LIN {X 0,Y 149.917,Z 380.311,A -85,B 0,C 180,E1 -25491.126,E2 -25491.126} C_VEL
LIN {X 0,Y 151.658,Z 366.446,A -85,B 0,C 180,E1 -25492.001,E2 -25492.001} C_VEL
LIN {X 0,Y 154.477,Z 327.485,A -85,B 0,C 180,E1 -25493.636,E2 -25493.636} C_VEL
LIN {X 0,Y 149.721,Z 315.229,A -85,B 0,C 180,E1 -25495.993,E2 -25495.993} C_VEL
LIN {X 0,Y 144.955,Z 306.325,A -85,B 0,C 180,E1 -25498.361,E2 -25498.361} C_VEL
LIN {X 0,Y 138.94,Z 296.328,A -85,B 0,C 180,E1 -25501.592,E2 -25501.592} C_VEL
LIN {X 0,Y 134.501,Z 289.677,A -85,B 0,C 180,E1 -25504.225,E2 -25504.225} C_VEL
LIN {X 0,Y 131.955,Z 285.984,A -85,B 0,C 180,E1 -25505.867,E2 -25505.867} C_VEL
LIN {X 0,Y 129.466,Z 282.342,A -85,B 0,C 180,E1 -25507.593,E2 -25507.593} C_VEL
LIN {X 0,Y 126.831,Z 279.366,A -85,B 0,C 180,E1 -25509.458,E2 -25509.458} C_VEL
LIN {X 0,Y 125.614,Z 277.233,A -85,B 0,C 180,E1 -25510.449,E2 -25510.449} C_VEL
LIN {X 0,Y 123.042,Z 275.019,A -85,B 0,C 180,E1 -25512.437,E2 -25512.437} C_VEL
LIN {X 0,Y 121.953,Z 272.605,A -85,B 0,C 180,E1 -25513.756,E2 -25513.756} C_VEL
LIN {X 0,Y 121.871,Z 271.831,A -85,B 0,C 180,E1 -25514.986,E2 -25514.986} C_VEL
LIN {X 0,Y 121.84,Z 271.763,A -85,B 0,C 180,E1 -25520.633,E2 -25520.633} C_VEL
LIN {X 0,Y 121.893,Z 271.784,A -85,B 0,C 180,E1 -25524.805,E2 -25524.805} C_VEL
LIN {X 0,Y 121.893,Z 271.751,A -85,B 0,C 180,E1 -25529.871,E2 -25529.871} C_VEL
LIN {X 0,Y 121.974,Z 271.79,A -85,B 0,C 180,E1 -25537.212,E2 -25537.212} C_VEL
LIN {X 0,Y 122.06,Z 271.721,A -85,B 0,C 180,E1 -25543.281,E2 -25543.281} C_VEL
LIN {X 0,Y 122.287,Z 271.749,A -85,B 0,C 180,E1 -25547.702,E2 -25547.702} C_VEL
LIN {X 0,Y 122.391,Z 271.714,A -85,B 0,C 180,E1 -25550.092,E2 -25550.092} C_VEL
LIN {X 0,Y 122.559,Z 271.673,A -85,B 0,C 180,E1 -25556.724,E2 -25556.724} C_VEL
LIN {X 0,Y 123.024,Z 271.658,A -85,B 0,C 180,E1 -25560.011,E2 -25560.011} C_VEL
LIN {X 0,Y 122.411,Z 271.686,A -85,B 0,C 180,E1 -25566.605,E2 -25566.605} C_VEL
LIN {X 0,Y 122.4,Z 271.735,A -85,B 0,C 180,E1 -25569.93,E2 -25569.93} C_VEL
LIN {X 0,Y 122.2,Z 271.727,A -85,B 0,C 180,E1 -25573.311,E2 -25573.311} C_VEL
LIN {X 0,Y 122.035,Z 271.781,A -85,B 0,C 180,E1 -25580.226,E2 -25580.226} C_VEL
LIN {X 0,Y 122.109,Z 271.951,A -85,B 0,C 180,E1 -25582.499,E2 -25582.499} C_VEL
LIN {X 0,Y 122.335,Z 273.222,A -85,B 0,C 180,E1 -25583.623,E2 -25583.623} C_VEL
LIN {X 0,Y 123.788,Z 275.687,A -85,B 0,C 180,E1 -25584.99,E2 -25584.99} C_VEL
LIN {X 0,Y 125.956,Z 277.488,A -85,B 0,C 180,E1 -25586.626,E2 -25586.626} C_VEL
LIN {X 0,Y 127.946,Z 280.764,A -85,B 0,C 180,E1 -25588.186,E2 -25588.186} C_VEL
LIN {X 0,Y 129.741,Z 282.697,A -85,B 0,C 180,E1 -25589.425,E2 -25589.425} C_VEL
LIN {X 0,Y 133.694,Z 288.444,A -85,B 0,C 180,E1 -25592.092,E2 -25592.092} C_VEL
LIN {X 0,Y 138.036,Z 294.974,A -85,B 0,C 180,E1 -25594.722,E2 -25594.722} C_VEL
LIN {X 0,Y 143.351,Z 303.799,A -85,B 0,C 180,E1 -25597.654,E2 -25597.654} C_VEL
LIN {X 0,Y 148.299,Z 314.843,A -85,B 0,C 180,E1 -25600.312,E2 -25600.312} C_VEL
LIN {X 0,Y 153.035,Z 327.628,A -85,B 0,C 180,E1 -25602.751,E2 -25602.751} C_VEL
LIN {X 0,Y 154.24,Z 331.13,A -85,B 0,C 180,E1 -25603.35,E2 -25603.35} C_VEL
LIN {X 0,Y 151.137,Z 374.069,A -85,B 0,C 180,E1 -25605.228,E2 -25605.228} C_VEL
LIN {X 0,Y 149.139,Z 387.318,A -85,B 0,C 180,E1 -25606.198,E2 -25606.198} C_VEL
LIN {X 0,Y 146.572,Z 399.758,A -85,B 0,C 180,E1 -25607.599,E2 -25607.599} C_VEL
LIN {X 0,Y 143.346,Z 411.689,A -85,B 0,C 180,E1 -25609.484,E2 -25609.484} C_VEL
LIN {X 0,Y 139.628,Z 423.169,A -85,B 0,C 180,E1 -25611.93,E2 -25611.93} C_VEL
LIN {X 0,Y 135.702,Z 433.514,A -85,B 0,C 180,E1 -25614.816,E2 -25614.816} C_VEL
LIN {X 0,Y 131.666,Z 443.348,A -85,B 0,C 180,E1 -25618.48,E2 -25618.48} C_VEL
LIN {X 0,Y 128.331,Z 451.168,A -85,B 0,C 180,E1 -25622.255,E2 -25622.255} C_VEL
LIN {X 0,Y 124.933,Z 458.531,A -85,B 0,C 180,E1 -25626.808,E2 -25626.808} C_VEL
LIN {X 0,Y 122.288,Z 464.413,A -85,B 0,C 180,E1 -25631.571,E2 -25631.571} C_VEL
LIN {X 0,Y 120.578,Z 469.032,A -85,B 0,C 180,E1 -25636.515,E2 -25636.515} C_VEL
LIN {X 0,Y 119.827,Z 471.455,A -85,B 0,C 180,E1 -25639.863,E2 -25639.863} C_VEL
LIN {X 0,Y 119.356,Z 473.43,A -85,B 0,C 180,E1 -25643.234,E2 -25643.234} C_VEL
LIN {X 0,Y 119.172,Z 474.984,A -85,B 0,C 180,E1 -25646.616,E2 -25646.616} C_VEL
LIN {X 0,Y 119.252,Z 476.091,A -85,B 0,C 180,E1 -25649.997,E2 -25649.997} C_VEL
LIN {X 0,Y 119.173,Z 476.77,A -85,B 0,C 180,E1 -25653.378,E2 -25653.378} C_VEL
LIN {X 0,Y 119.89,Z 476.987,A -85,B 0,C 180,E1 -25660.126,E2 -25660.126} C_VEL
LIN {X 0,Y 120.731,Z 476.514,A -85,B 0,C 180,E1 -25663.462,E2 -25663.462} C_VEL
LIN {X 0,Y 123.396,Z 474.35,A -85,B 0,C 180,E1 -25669.979,E2 -25669.979} C_VEL
LIN {X 0,Y 126.498,Z 471.676,A -85,B 0,C 180,E1 -25674.622,E2 -25674.622} C_VEL
LIN {X 0,Y 130.853,Z 467.562,A -85,B 0,C 180,E1 -25679.473,E2 -25679.473} C_VEL
LIN {X 0,Y 136.528,Z 461.498,A -85,B 0,C 180,E1 -25684.485,E2 -25684.485} C_VEL
LIN {X 0,Y 141.954,Z 455.109,A -85,B 0,C 180,E1 -25688.23,E2 -25688.23} C_VEL
LIN {X 0,Y 143.742,Z 452.844,A -85,B 0,C 180,E1 -25689.335,E2 -25689.335} C_VEL
LIN {X 0,Y 145.909,Z 449.452,A -85,B 0,C 180,E1 -25691.051,E2 -25691.051} C_VEL
LIN {X 0,Y 148.208,Z 443.627,A -85,B 0,C 180,E1 -25694.05,E2 -25694.05} C_VEL
LIN {X 0,Y 150.646,Z 437.293,A -85,B 0,C 180,E1 -25696.796,E2 -25696.796} C_VEL
LIN {X 0,Y 152.93,Z 433.024,A -85,B 0,C 180,E1 -25698.077,E2 -25698.077} C_VEL
LIN {X 0,Y 158.845,Z 422.424,A -85,B 0,C 180,E1 -25700.238,E2 -25700.238} C_VEL
LIN {X 0,Y 164.023,Z 411.245,A -85,B 0,C 180,E1 -25701.932,E2 -25701.932} C_VEL
LIN {X 0,Y 168.444,Z 399.218,A -85,B 0,C 180,E1 -25703.309,E2 -25703.309} C_VEL
LIN {X 0,Y 171.869,Z 387.049,A -85,B 0,C 180,E1 -25704.268,E2 -25704.268} C_VEL
LIN {X 0,Y 174.526,Z 373.628,A -85,B 0,C 180,E1 -25704.952,E2 -25704.952} C_VEL
LIN {X 0,Y 176.895,Z 350.528,A -85,B 0,C 180,E1 -25705.791,E2 -25705.791} C_VEL
LIN {X 0,Y 174.129,Z 342.792,A -85,B 0,C 180,E1 -25708.604,E2 -25708.604} C_VEL
LIN {X 0,Y 171.468,Z 336.339,A -85,B 0,C 180,E1 -25711.689,E2 -25711.689} C_VEL
LIN {X 0,Y 170.136,Z 333.483,A -85,B 0,C 180,E1 -25713.465,E2 -25713.465} C_VEL
LIN {X 0,Y 168.525,Z 330.627,A -85,B 0,C 180,E1 -25715.864,E2 -25715.864} C_VEL
LIN {X 0,Y 166.557,Z 327.038,A -85,B 0,C 180,E1 -25719.732,E2 -25719.732} C_VEL
LIN {X 0,Y 164.734,Z 324.215,A -85,B 0,C 180,E1 -25727.052,E2 -25727.052} C_VEL
LIN {X 0,Y 164.785,Z 323.798,A -85,B 0,C 180,E1 -25730.169,E2 -25730.169} C_VEL
LIN {X 0,Y 166.586,Z 326.483,A -85,B 0,C 180,E1 -25737.423,E2 -25737.423} C_VEL
LIN {X 0,Y 168.586,Z 330.291,A -85,B 0,C 180,E1 -25741.404,E2 -25741.404} C_VEL
LIN {X 0,Y 170.651,Z 333.974,A -85,B 0,C 180,E1 -25744.408,E2 -25744.408} C_VEL
LIN {X 0,Y 173.991,Z 340.469,A -85,B 0,C 180,E1 -25748.266,E2 -25748.266} C_VEL
LIN {X 0,Y 175.805,Z 344.628,A -85,B 0,C 180,E1 -25750.115,E2 -25750.115} C_VEL
LIN {X 0,Y 177.089,Z 348.243,A -85,B 0,C 180,E1 -25751.363,E2 -25751.363} C_VEL
LIN {X 0,Y 174.518,Z 372.291,A -85,B 0,C 180,E1 -25752.203,E2 -25752.203} C_VEL
LIN {X 0,Y 172.102,Z 384.595,A -85,B 0,C 180,E1 -25752.859,E2 -25752.859} C_VEL
LIN {X 0,Y 168.746,Z 396.829,A -85,B 0,C 180,E1 -25753.859,E2 -25753.859} C_VEL
LIN {X 0,Y 164.693,Z 408.226,A -85,B 0,C 180,E1 -25755.201,E2 -25755.201} C_VEL
LIN {X 0,Y 159.734,Z 419.22,A -85,B 0,C 180,E1 -25756.882,E2 -25756.882} C_VEL
LIN {X 0,Y 154.191,Z 429.462,A -85,B 0,C 180,E1 -25758.962,E2 -25758.962} C_VEL
LIN {X 0,Y 148.873,Z 437.871,A -85,B 0,C 180,E1 -25761.196,E2 -25761.196} C_VEL
LIN {X 0,Y 142.551,Z 446.547,A -85,B 0,C 180,E1 -25764.212,E2 -25764.212} C_VEL
LIN {X 0,Y 136.628,Z 453.681,A -85,B 0,C 180,E1 -25767.565,E2 -25767.565} C_VEL
LIN {X 0,Y 129.941,Z 460.795,A -85,B 0,C 180,E1 -25772.199,E2 -25772.199} C_VEL
LIN {X 0,Y 123.977,Z 466.358,A -85,B 0,C 180,E1 -25777.479,E2 -25777.479} C_VEL
LIN {X 0,Y 119.536,Z 470.003,A -85,B 0,C 180,E1 -25782.704,E2 -25782.704} C_VEL
LIN {X 0,Y 116.059,Z 472.435,A -85,B 0,C 180,E1 -25788.237,E2 -25788.237} C_VEL
LIN {X 0,Y 113.852,Z 473.647,A -85,B 0,C 180,E1 -25793.345,E2 -25793.345} C_VEL
LIN {X 0,Y 112.133,Z 473.944,A -85,B 0,C 180,E1 -25799.911,E2 -25799.911} C_VEL
LIN {X 0,Y 111.656,Z 473.511,A -85,B 0,C 180,E1 -25803.861,E2 -25803.861} C_VEL
LIN {X 0,Y 111.688,Z 471.595,A -85,B 0,C 180,E1 -25810.67,E2 -25810.67} C_VEL
LIN {X 0,Y 112.749,Z 468.214,A -85,B 0,C 180,E1 -25817.402,E2 -25817.402} C_VEL
LIN {X 0,Y 114.461,Z 464.126,A -85,B 0,C 180,E1 -25822.949,E2 -25822.949} C_VEL
LIN {X 0,Y 116.793,Z 458.839,A -85,B 0,C 180,E1 -25828.279,E2 -25828.279} C_VEL
LIN {X 0,Y 120.046,Z 452.098,A -85,B 0,C 180,E1 -25833.359,E2 -25833.359} C_VEL
LIN {X 0,Y 124.034,Z 443.668,A -85,B 0,C 180,E1 -25838.146,E2 -25838.146} C_VEL
LIN {X 0,Y 127.929,Z 435.024,A -85,B 0,C 180,E1 -25841.891,E2 -25841.891} C_VEL
LIN {X 0,Y 131.791,Z 425.809,A -85,B 0,C 180,E1 -25844.967,E2 -25844.967} C_VEL
LIN {X 0,Y 135.727,Z 415.062,A -85,B 0,C 180,E1 -25847.713,E2 -25847.713} C_VEL
LIN {X 0,Y 139.216,Z 403.697,A -85,B 0,C 180,E1 -25849.925,E2 -25849.925} C_VEL
LIN {X 0,Y 142.282,Z 391.091,A -85,B 0,C 180,E1 -25851.746,E2 -25851.746} C_VEL
LIN {X 0,Y 144.771,Z 377.58,A -85,B 0,C 180,E1 -25853.038,E2 -25853.038} C_VEL
LIN {X 0,Y 146.278,Z 364.752,A -85,B 0,C 180,E1 -25853.806,E2 -25853.806} C_VEL
LIN {X 0,Y 148.904,Z 329.221,A -85,B 0,C 180,E1 -25855.326,E2 -25855.326} C_VEL
LIN {X 0,Y 144.595,Z 318.262,A -85,B 0,C 180,E1 -25857.637,E2 -25857.637} C_VEL
LIN {X 0,Y 139.163,Z 308.178,A -85,B 0,C 180,E1 -25860.558,E2 -25860.558} C_VEL
LIN {X 0,Y 133.577,Z 298.915,A -85,B 0,C 180,E1 -25863.891,E2 -25863.891} C_VEL
LIN {X 0,Y 128.421,Z 291.313,A -85,B 0,C 180,E1 -25867.331,E2 -25867.331} C_VEL
LIN {X 0,Y 125.856,Z 287.671,A -85,B 0,C 180,E1 -25869.228,E2 -25869.228} C_VEL
LIN {X 0,Y 123.261,Z 284.164,A -85,B 0,C 180,E1 -25871.279,E2 -25871.279} C_VEL
LIN {X 0,Y 122.402,Z 283.086,A -85,B 0,C 180,E1 -25871.994,E2 -25871.994} C_VEL
LIN {X 0,Y 119.918,Z 280.305,A -85,B 0,C 180,E1 -25874.161,E2 -25874.161} C_VEL
LIN {X 0,Y 118.797,Z 278.232,A -85,B 0,C 180,E1 -25875.317,E2 -25875.317} C_VEL
LIN {X 0,Y 116.391,Z 276.344,A -85,B 0,C 180,E1 -25877.624,E2 -25877.624} C_VEL
LIN {X 0,Y 114.926,Z 273.384,A -85,B 0,C 180,E1 -25879.782,E2 -25879.782} C_VEL
LIN {X 0,Y 114.783,Z 272.721,A -85,B 0,C 180,E1 -25881.144,E2 -25881.144} C_VEL
LIN {X 0,Y 114.795,Z 272.679,A -85,B 0,C 180,E1 -25886.58,E2 -25886.58} C_VEL
LIN {X 0,Y 114.806,Z 272.629,A -85,B 0,C 180,E1 -25890.692,E2 -25890.692} C_VEL
LIN {X 0,Y 114.893,Z 272.673,A -85,B 0,C 180,E1 -25896.576,E2 -25896.576} C_VEL
LIN {X 0,Y 114.963,Z 272.603,A -85,B 0,C 180,E1 -25902.215,E2 -25902.215} C_VEL
LIN {X 0,Y 115.306,Z 272.605,A -85,B 0,C 180,E1 -25909.476,E2 -25909.476} C_VEL
LIN {X 0,Y 115.485,Z 272.55,A -85,B 0,C 180,E1 -25916.523,E2 -25916.523} C_VEL
LIN {X 0,Y 115.976,Z 272.536,A -85,B 0,C 180,E1 -25920.012,E2 -25920.012} C_VEL
LIN {X 0,Y 115.354,Z 272.567,A -85,B 0,C 180,E1 -25927.011,E2 -25927.011} C_VEL
LIN {X 0,Y 115.215,Z 272.604,A -85,B 0,C 180,E1 -25932.572,E2 -25932.572} C_VEL
LIN {X 0,Y 115.072,Z 272.837,A -85,B 0,C 180,E1 -25936.42,E2 -25936.42} C_VEL
LIN {X 0,Y 115.35,Z 274.101,A -85,B 0,C 180,E1 -25937.863,E2 -25937.863} C_VEL
LIN {X 0,Y 116.774,Z 276.567,A -85,B 0,C 180,E1 -25939.571,E2 -25939.571} C_VEL
LIN {X 0,Y 119.245,Z 278.524,A -85,B 0,C 180,E1 -25941.917,E2 -25941.917} C_VEL
LIN {X 0,Y 121.112,Z 281.678,A -85,B 0,C 180,E1 -25943.742,E2 -25943.742} C_VEL
LIN {X 0,Y 123.21,Z 283.867,A -85,B 0,C 180,E1 -25945.482,E2 -25945.482} C_VEL
LIN {X 0,Y 125.712,Z 287.403,A -85,B 0,C 180,E1 -25947.483,E2 -25947.483} C_VEL
LIN {X 0,Y 127.202,Z 289.451,A -85,B 0,C 180,E1 -25948.601,E2 -25948.601} C_VEL
LIN {X 0,Y 130.687,Z 294.469,A -85,B 0,C 180,E1 -25951.05,E2 -25951.05} C_VEL
LIN {X 0,Y 136.464,Z 303.687,A -85,B 0,C 180,E1 -25954.716,E2 -25954.716} C_VEL
LIN {X 0,Y 139.996,Z 310.198,A -85,B 0,C 180,E1 -25956.777,E2 -25956.777} C_VEL
LIN {X 0,Y 145.15,Z 322.701,A -85,B 0,C 180,E1 -25959.72,E2 -25959.72} C_VEL
LIN {X 0,Y 148.753,Z 333.117,A -85,B 0,C 180,E1 -25961.715,E2 -25961.715} C_VEL
LIN {X 0,Y 145.583,Z 374.151,A -85,B 0,C 180,E1 -25963.534,E2 -25963.534} C_VEL
LIN {X 0,Y 143.513,Z 387.259,A -85,B 0,C 180,E1 -25964.506,E2 -25964.506} C_VEL
LIN {X 0,Y 140.849,Z 399.691,A -85,B 0,C 180,E1 -25965.934,E2 -25965.934} C_VEL
LIN {X 0,Y 137.486,Z 411.614,A -85,B 0,C 180,E1 -25967.859,E2 -25967.859} C_VEL
LIN {X 0,Y 133.601,Z 423.09,A -85,B 0,C 180,E1 -25970.367,E2 -25970.367} C_VEL
LIN {X 0,Y 129.491,Z 433.431,A -85,B 0,C 180,E1 -25973.341,E2 -25973.341} C_VEL
LIN {X 0,Y 125.432,Z 442.85,A -85,B 0,C 180,E1 -25976.955,E2 -25976.955} C_VEL
LIN {X 0,Y 122.059,Z 450.396,A -85,B 0,C 180,E1 -25980.695,E2 -25980.695} C_VEL
LIN {X 0,Y 118.421,Z 457.879,A -85,B 0,C 180,E1 -25985.451,E2 -25985.451} C_VEL
LIN {X 0,Y 115.537,Z 463.867,A -85,B 0,C 180,E1 -25990.451,E2 -25990.451} C_VEL
LIN {X 0,Y 113.667,Z 468.589,A -85,B 0,C 180,E1 -25995.678,E2 -25995.678} C_VEL
LIN {X 0,Y 112.514,Z 472.165,A -85,B 0,C 180,E1 -26001.013,E2 -26001.013} C_VEL
LIN {X 0,Y 112.08,Z 474.707,A -85,B 0,C 180,E1 -26006.402,E2 -26006.402} C_VEL
LIN {X 0,Y 112.156,Z 475.888,A -85,B 0,C 180,E1 -26009.997,E2 -26009.997} C_VEL
LIN {X 0,Y 112.081,Z 476.612,A -85,B 0,C 180,E1 -26013.592,E2 -26013.592} C_VEL
LIN {X 0,Y 112.902,Z 476.907,A -85,B 0,C 180,E1 -26020.76,E2 -26020.76} C_VEL
LIN {X 0,Y 113.812,Z 476.49,A -85,B 0,C 180,E1 -26024.297,E2 -26024.297} C_VEL
LIN {X 0,Y 115.101,Z 475.666,A -85,B 0,C 180,E1 -26027.773,E2 -26027.773} C_VEL
LIN {X 0,Y 116.721,Z 474.438,A -85,B 0,C 180,E1 -26031.175,E2 -26031.175} C_VEL
LIN {X 0,Y 121.378,Z 470.796,A -85,B 0,C 180,E1 -26037.591,E2 -26037.591} C_VEL
LIN {X 0,Y 125.754,Z 466.888,A -85,B 0,C 180,E1 -26042.064,E2 -26042.064} C_VEL
LIN {X 0,Y 130.741,Z 461.895,A -85,B 0,C 180,E1 -26046.246,E2 -26046.246} C_VEL
LIN {X 0,Y 136.461,Z 455.652,A -85,B 0,C 180,E1 -26050.07,E2 -26050.07} C_VEL
LIN {X 0,Y 142.8,Z 447.875,A -85,B 0,C 180,E1 -26053.549,E2 -26053.549} C_VEL
LIN {X 0,Y 149.607,Z 438.265,A -85,B 0,C 180,E1 -26056.726,E2 -26056.726} C_VEL
LIN {X 0,Y 152.93,Z 433.024,A -85,B 0,C 180,E1 -26058.077,E2 -26058.077} C_VEL
LIN {X 0,Y 155.209,Z 428.626,A -85,B 0,C 180,E1 -26059.282,E2 -26059.282} C_VEL
LIN {X 0,Y 157.669,Z 421.297,A -85,B 0,C 180,E1 -26061.563,E2 -26061.563} C_VEL
LIN {X 0,Y 159.898,Z 413.531,A -85,B 0,C 180,E1 -26063.626,E2 -26063.626} C_VEL
LIN {X 0,Y 161.717,Z 408.455,A -85,B 0,C 180,E1 -26064.475,E2 -26064.475} C_VEL
LIN {X 0,Y 166.123,Z 396.063,A -85,B 0,C 180,E1 -26065.754,E2 -26065.754} C_VEL
LIN {X 0,Y 169.642,Z 383.168,A -85,B 0,C 180,E1 -26066.625,E2 -26066.625} C_VEL
LIN {X 0,Y 171.89,Z 370.23,A -85,B 0,C 180,E1 -26067.222,E2 -26067.222} C_VEL
LIN {X 0,Y 173.598,Z 353.693,A -85,B 0,C 180,E1 -26067.801,E2 -26067.801} C_VEL
LIN {X 0,Y 171.078,Z 346.284,A -85,B 0,C 180,E1 -26070.757,E2 -26070.757} C_VEL
LIN {X 0,Y 168.825,Z 340.5,A -85,B 0,C 180,E1 -26073.847,E2 -26073.847} C_VEL
LIN {X 0,Y 166.972,Z 337.147,A -85,B 0,C 180,E1 -26076.764,E2 -26076.764} C_VEL
LIN {X 0,Y 165.208,Z 333.639,A -85,B 0,C 180,E1 -26080.684,E2 -26080.684} C_VEL
LIN {X 0,Y 163.761,Z 331.034,A -85,B 0,C 180,E1 -26087.988,E2 -26087.988} C_VEL
LIN {X 0,Y 163.867,Z 331.008,A -85,B 0,C 180,E1 -26090.536,E2 -26090.536} C_VEL
LIN {X 0,Y 165.36,Z 333.254,A -85,B 0,C 180,E1 -26096.778,E2 -26096.778} C_VEL
LIN {X 0,Y 167.707,Z 337.979,A -85,B 0,C 180,E1 -26101.628,E2 -26101.628} C_VEL
LIN {X 0,Y 169.661,Z 341.982,A -85,B 0,C 180,E1 -26104.537,E2 -26104.537} C_VEL
LIN {X 0,Y 172.173,Z 347.158,A -85,B 0,C 180,E1 -26107.552,E2 -26107.552} C_VEL
LIN {X 0,Y 173.612,Z 350.795,A -85,B 0,C 180,E1 -26109.135,E2 -26109.135} C_VEL
LIN {X 0,Y 173.827,Z 351.507,A -85,B 0,C 180,E1 -26109.379,E2 -26109.379} C_VEL
LIN {X 0,Y 171.331,Z 373.134,A -85,B 0,C 180,E1 -26110.122,E2 -26110.122} C_VEL
LIN {X 0,Y 168.814,Z 385.293,A -85,B 0,C 180,E1 -26110.767,E2 -26110.767} C_VEL
LIN {X 0,Y 165.125,Z 397.939,A -85,B 0,C 180,E1 -26111.798,E2 -26111.798} C_VEL
LIN {X 0,Y 160.24,Z 410.64,A -85,B 0,C 180,E1 -26113.311,E2 -26113.311} C_VEL
LIN {X 0,Y 154.705,Z 422.04,A -85,B 0,C 180,E1 -26115.137,E2 -26115.137} C_VEL
LIN {X 0,Y 148.822,Z 431.947,A -85,B 0,C 180,E1 -26117.249,E2 -26117.249} C_VEL
LIN {X 0,Y 142.118,Z 441.572,A -85,B 0,C 180,E1 -26120.026,E2 -26120.026} C_VEL
LIN {X 0,Y 135.661,Z 449.573,A -85,B 0,C 180,E1 -26123.148,E2 -26123.148} C_VEL
LIN {X 0,Y 129.633,Z 456.128,A -85,B 0,C 180,E1 -26126.598,E2 -26126.598} C_VEL
LIN {X 0,Y 123.154,Z 462.318,A -85,B 0,C 180,E1 -26131.135,E2 -26131.135} C_VEL
LIN {X 0,Y 117.771,Z 466.853,A -85,B 0,C 180,E1 -26135.857,E2 -26135.857} C_VEL
LIN {X 0,Y 112.809,Z 470.549,A -85,B 0,C 180,E1 -26141.622,E2 -26141.622} C_VEL
LIN {X 0,Y 110.245,Z 472.203,A -85,B 0,C 180,E1 -26145.478,E2 -26145.478} C_VEL
LIN {X 0,Y 107.155,Z 473.743,A -85,B 0,C 180,E1 -26151.887,E2 -26151.887} C_VEL
LIN {X 0,Y 105.413,Z 474.1,A -85,B 0,C 180,E1 -26157.771,E2 -26157.771} C_VEL
LIN {X 0,Y 104.727,Z 473.762,A -85,B 0,C 180,E1 -26161.985,E2 -26161.985} C_VEL
LIN {X 0,Y 104.415,Z 472.99,A -85,B 0,C 180,E1 -26166.185,E2 -26166.185} C_VEL
LIN {X 0,Y 104.572,Z 471.717,A -85,B 0,C 180,E1 -26170.368,E2 -26170.368} C_VEL
LIN {X 0,Y 105.399,Z 468.945,A -85,B 0,C 180,E1 -26176.507,E2 -26176.507} C_VEL
LIN {X 0,Y 107.079,Z 465.06,A -85,B 0,C 180,E1 -26182.46,E2 -26182.46} C_VEL
LIN {X 0,Y 109.414,Z 459.992,A -85,B 0,C 180,E1 -26188.163,E2 -26188.163} C_VEL
LIN {X 0,Y 112.68,Z 453.558,A -85,B 0,C 180,E1 -26193.579,E2 -26193.579} C_VEL
LIN {X 0,Y 116.748,Z 445.487,A -85,B 0,C 180,E1 -26198.658,E2 -26198.658} C_VEL
LIN {X 0,Y 120.75,Z 437.176,A -85,B 0,C 180,E1 -26202.61,E2 -26202.61} C_VEL
LIN {X 0,Y 125.314,Z 426.978,A -85,B 0,C 180,E1 -26206.288,E2 -26206.288} C_VEL
LIN {X 0,Y 129.266,Z 416.931,A -85,B 0,C 180,E1 -26209.042,E2 -26209.042} C_VEL
LIN {X 0,Y 132.911,Z 405.988,A -85,B 0,C 180,E1 -26211.32,E2 -26211.32} C_VEL
LIN {X 0,Y 136.328,Z 392.896,A -85,B 0,C 180,E1 -26213.35,E2 -26213.35} C_VEL
LIN {X 0,Y 138.914,Z 380.37,A -85,B 0,C 180,E1 -26214.66,E2 -26214.66} C_VEL
LIN {X 0,Y 140.641,Z 367.677,A -85,B 0,C 180,E1 -26215.508,E2 -26215.508} C_VEL
LIN {X 0,Y 143.513,Z 331.247,A -85,B 0,C 180,E1 -26217.109,E2 -26217.109} C_VEL
LIN {X 0,Y 139.947,Z 322.152,A -85,B 0,C 180,E1 -26219.157,E2 -26219.157} C_VEL
LIN {X 0,Y 134.956,Z 312.647,A -85,B 0,C 180,E1 -26222.07,E2 -26222.07} C_VEL
LIN {X 0,Y 129.746,Z 303.794,A -85,B 0,C 180,E1 -26225.431,E2 -26225.431} C_VEL
LIN {X 0,Y 125.285,Z 296.99,A -85,B 0,C 180,E1 -26228.634,E2 -26228.634} C_VEL
LIN {X 0,Y 122.561,Z 293.159,A -85,B 0,C 180,E1 -26230.785,E2 -26230.785} C_VEL
LIN {X 0,Y 119.742,Z 289.21,A -85,B 0,C 180,E1 -26233.239,E2 -26233.239} C_VEL
LIN {X 0,Y 117.208,Z 286.087,A -85,B 0,C 180,E1 -26235.636,E2 -26235.636} C_VEL
LIN {X 0,Y 116.356,Z 284.597,A -85,B 0,C 180,E1 -26236.561,E2 -26236.561} C_VEL
LIN {X 0,Y 113.858,Z 282.238,A -85,B 0,C 180,E1 -26239.18,E2 -26239.18} C_VEL
LIN {X 0,Y 112.264,Z 279.369,A -85,B 0,C 180,E1 -26241.26,E2 -26241.26} C_VEL
LIN {X 0,Y 109.315,Z 277.263,A -85,B 0,C 180,E1 -26245.196,E2 -26245.196} C_VEL
LIN {X 0,Y 107.91,Z 274.351,A -85,B 0,C 180,E1 -26248.162,E2 -26248.162} C_VEL
LIN {X 0,Y 107.764,Z 273.577,A -85,B 0,C 180,E1 -26250.733,E2 -26250.733} C_VEL
LIN {X 0,Y 107.861,Z 273.548,A -85,B 0,C 180,E1 -26257.001,E2 -26257.001} C_VEL
LIN {X 0,Y 107.858,Z 273.491,A -85,B 0,C 180,E1 -26261,E2 -26261} C_VEL
LIN {X 0,Y 108.224,Z 273.498,A -85,B 0,C 180,E1 -26268.779,E2 -26268.779} C_VEL
LIN {X 0,Y 108.287,Z 273.437,A -85,B 0,C 180,E1 -26272.555,E2 -26272.555} C_VEL
LIN {X 0,Y 108.902,Z 273.416,A -85,B 0,C 180,E1 -26280.013,E2 -26280.013} C_VEL
LIN {X 0,Y 108.293,Z 273.656,A -85,B 0,C 180,E1 -26287.939,E2 -26287.939} C_VEL
LIN {X 0,Y 108.611,Z 274.943,A -85,B 0,C 180,E1 -26290.145,E2 -26290.145} C_VEL
LIN {X 0,Y 110.026,Z 277.458,A -85,B 0,C 180,E1 -26292.608,E2 -26292.608} C_VEL
LIN {X 0,Y 112.693,Z 279.681,A -85,B 0,C 180,E1 -26296.078,E2 -26296.078} C_VEL
LIN {X 0,Y 114.499,Z 282.825,A -85,B 0,C 180,E1 -26298.347,E2 -26298.347} C_VEL
LIN {X 0,Y 116.809,Z 284.994,A -85,B 0,C 180,E1 -26300.712,E2 -26300.712} C_VEL
LIN {X 0,Y 119.069,Z 288.379,A -85,B 0,C 180,E1 -26302.976,E2 -26302.976} C_VEL
LIN {X 0,Y 120.476,Z 289.98,A -85,B 0,C 180,E1 -26304.227,E2 -26304.227} C_VEL
LIN {X 0,Y 124.461,Z 295.65,A -85,B 0,C 180,E1 -26307.542,E2 -26307.542} C_VEL
LIN {X 0,Y 128.367,Z 301.526,A -85,B 0,C 180,E1 -26310.437,E2 -26310.437} C_VEL
LIN {X 0,Y 134.288,Z 311.608,A -85,B 0,C 180,E1 -26314.361,E2 -26314.361} C_VEL
LIN {X 0,Y 138.192,Z 320.508,A -85,B 0,C 180,E1 -26316.82,E2 -26316.82} C_VEL
LIN {X 0,Y 142.503,Z 332.46,A -85,B 0,C 180,E1 -26319.429,E2 -26319.429} C_VEL
LIN {X 0,Y 143.327,Z 334.933,A -85,B 0,C 180,E1 -26319.918,E2 -26319.918} C_VEL
LIN {X 0,Y 140.209,Z 373.782,A -85,B 0,C 180,E1 -26321.673,E2 -26321.673} C_VEL
LIN {X 0,Y 138.023,Z 387.2,A -85,B 0,C 180,E1 -26322.678,E2 -26322.678} C_VEL
LIN {X 0,Y 135.254,Z 399.624,A -85,B 0,C 180,E1 -26324.131,E2 -26324.131} C_VEL
LIN {X 0,Y 131.733,Z 411.534,A -85,B 0,C 180,E1 -26326.085,E2 -26326.085} C_VEL
LIN {X 0,Y 127.682,Z 423.01,A -85,B 0,C 180,E1 -26328.658,E2 -26328.658} C_VEL
LIN {X 0,Y 123.379,Z 433.349,A -85,B 0,C 180,E1 -26331.719,E2 -26331.719} C_VEL
LIN {X 0,Y 118.769,Z 443.47,A -85,B 0,C 180,E1 -26335.794,E2 -26335.794} C_VEL
LIN {X 0,Y 114.45,Z 452.358,A -85,B 0,C 180,E1 -26340.574,E2 -26340.574} C_VEL
LIN {X 0,Y 110.854,Z 459.428,A -85,B 0,C 180,E1 -26345.661,E2 -26345.661} C_VEL
LIN {X 0,Y 108.031,Z 465.061,A -85,B 0,C 180,E1 -26351.015,E2 -26351.015} C_VEL
LIN {X 0,Y 106.277,Z 469.482,A -85,B 0,C 180,E1 -26356.614,E2 -26356.614} C_VEL
LIN {X 0,Y 105.255,Z 472.793,A -85,B 0,C 180,E1 -26362.323,E2 -26362.323} C_VEL
LIN {X 0,Y 104.985,Z 474.427,A -85,B 0,C 180,E1 -26366.158,E2 -26366.158} C_VEL
LIN {X 0,Y 105.055,Z 475.655,A -85,B 0,C 180,E1 -26369.997,E2 -26369.997} C_VEL
LIN {X 0,Y 104.986,Z 476.452,A -85,B 0,C 180,E1 -26373.835,E2 -26373.835} C_VEL
LIN {X 0,Y 105.915,Z 476.829,A -85,B 0,C 180,E1 -26381.479,E2 -26381.479} C_VEL
LIN {X 0,Y 108.334,Z 475.706,A -85,B 0,C 180,E1 -26388.924,E2 -26388.924} C_VEL
LIN {X 0,Y 110.107,Z 474.534,A -85,B 0,C 180,E1 -26392.515,E2 -26392.515} C_VEL
LIN {X 0,Y 115.138,Z 470.981,A -85,B 0,C 180,E1 -26399.226,E2 -26399.226} C_VEL
LIN {X 0,Y 119.781,Z 467.17,A -85,B 0,C 180,E1 -26403.872,E2 -26403.872} C_VEL
LIN {X 0,Y 125.091,Z 462.291,A -85,B 0,C 180,E1 -26408.167,E2 -26408.167} C_VEL
LIN {X 0,Y 131.132,Z 456.187,A -85,B 0,C 180,E1 -26412.058,E2 -26412.058} C_VEL
LIN {X 0,Y 137.784,Z 448.626,A -85,B 0,C 180,E1 -26415.566,E2 -26415.566} C_VEL
LIN {X 0,Y 144.87,Z 439.188,A -85,B 0,C 180,E1 -26418.755,E2 -26418.755} C_VEL
LIN {X 0,Y 151.249,Z 429.466,A -85,B 0,C 180,E1 -26421.102,E2 -26421.102} C_VEL
LIN {X 0,Y 157.127,Z 418.663,A -85,B 0,C 180,E1 -26423.08,E2 -26423.08} C_VEL
LIN {X 0,Y 161.717,Z 408.455,A -85,B 0,C 180,E1 -26424.475,E2 -26424.475} C_VEL
LIN {X 0,Y 163.43,Z 403.268,A -85,B 0,C 180,E1 -26425.266,E2 -26425.266} C_VEL
LIN {X 0,Y 165.088,Z 394.763,A -85,B 0,C 180,E1 -26426.96,E2 -26426.96} C_VEL
LIN {X 0,Y 166.36,Z 386.008,A -85,B 0,C 180,E1 -26428.476,E2 -26428.476} C_VEL
LIN {X 0,Y 167.38,Z 380.412,A -85,B 0,C 180,E1 -26428.985,E2 -26428.985} C_VEL
LIN {X 0,Y 169.547,Z 366.781,A -85,B 0,C 180,E1 -26429.555,E2 -26429.555} C_VEL
LIN {X 0,Y 170.546,Z 357.001,A -85,B 0,C 180,E1 -26429.892,E2 -26429.892} C_VEL
LIN {X 0,Y 168.536,Z 350.777,A -85,B 0,C 180,E1 -26432.604,E2 -26432.604} C_VEL
LIN {X 0,Y 166.955,Z 346.463,A -85,B 0,C 180,E1 -26435.097,E2 -26435.097} C_VEL
LIN {X 0,Y 165.551,Z 343.752,A -85,B 0,C 180,E1 -26437.53,E2 -26437.53} C_VEL
LIN {X 0,Y 164.009,Z 340.434,A -85,B 0,C 180,E1 -26441.341,E2 -26441.341} C_VEL
LIN {X 0,Y 162.822,Z 337.948,A -85,B 0,C 180,E1 -26448.753,E2 -26448.753} C_VEL
LIN {X 0,Y 162.918,Z 338.115,A -85,B 0,C 180,E1 -26450.48,E2 -26450.48} C_VEL
LIN {X 0,Y 164.244,Z 340.322,A -85,B 0,C 180,E1 -26456.414,E2 -26456.414} C_VEL
LIN {X 0,Y 166.289,Z 344.697,A -85,B 0,C 180,E1 -26460.967,E2 -26460.967} C_VEL
LIN {X 0,Y 167.935,Z 348.304,A -85,B 0,C 180,E1 -26463.611,E2 -26463.611} C_VEL
LIN {X 0,Y 170.15,Z 353.271,A -85,B 0,C 180,E1 -26466.543,E2 -26466.543} C_VEL
LIN {X 0,Y 170.77,Z 354.801,A -85,B 0,C 180,E1 -26467.281,E2 -26467.281} C_VEL
LIN {X 0,Y 168.473,Z 373.679,A -85,B 0,C 180,E1 -26467.938,E2 -26467.938} C_VEL
LIN {X 0,Y 165.927,Z 385.466,A -85,B 0,C 180,E1 -26468.535,E2 -26468.535} C_VEL
LIN {X 0,Y 162.607,Z 396.684,A -85,B 0,C 180,E1 -26469.403,E2 -26469.403} C_VEL
LIN {X 0,Y 158.278,Z 408.082,A -85,B 0,C 180,E1 -26470.661,E2 -26470.661} C_VEL
LIN {X 0,Y 152.842,Z 419.313,A -85,B 0,C 180,E1 -26472.293,E2 -26472.293} C_VEL
LIN {X 0,Y 146.346,Z 430.308,A -85,B 0,C 180,E1 -26474.439,E2 -26474.439} C_VEL
LIN {X 0,Y 139.623,Z 439.826,A -85,B 0,C 180,E1 -26476.996,E2 -26476.996} C_VEL
LIN {X 0,Y 132.749,Z 448.122,A -85,B 0,C 180,E1 -26480.003,E2 -26480.003} C_VEL
LIN {X 0,Y 125.666,Z 455.547,A -85,B 0,C 180,E1 -26483.713,E2 -26483.713} C_VEL
LIN {X 0,Y 118.602,Z 461.98,A -85,B 0,C 180,E1 -26488.284,E2 -26488.284} C_VEL
LIN {X 0,Y 112.947,Z 466.461,A -85,B 0,C 180,E1 -26492.864,E2 -26492.864} C_VEL
LIN {X 0,Y 107.657,Z 470.126,A -85,B 0,C 180,E1 -26498.435,E2 -26498.435} C_VEL
LIN {X 0,Y 104.707,Z 471.896,A -85,B 0,C 180,E1 -26502.416,E2 -26502.416} C_VEL
LIN {X 0,Y 102.221,Z 473.171,A -85,B 0,C 180,E1 -26506.57,E2 -26506.57} C_VEL
LIN {X 0,Y 100.291,Z 473.915,A -85,B 0,C 180,E1 -26510.904,E2 -26510.904} C_VEL
LIN {X 0,Y 98.843,Z 474.208,A -85,B 0,C 180,E1 -26515.336,E2 -26515.336} C_VEL
LIN {X 0,Y 97.913,Z 474.011,A -85,B 0,C 180,E1 -26519.842,E2 -26519.842} C_VEL
LIN {X 0,Y 97.379,Z 473.332,A -85,B 0,C 180,E1 -26524.344,E2 -26524.344} C_VEL
LIN {X 0,Y 97.402,Z 471.953,A -85,B 0,C 180,E1 -26529.673,E2 -26529.673} C_VEL
LIN {X 0,Y 98.068,Z 469.638,A -85,B 0,C 180,E1 -26535.477,E2 -26535.477} C_VEL
LIN {X 0,Y 99.662,Z 465.963,A -85,B 0,C 180,E1 -26541.896,E2 -26541.896} C_VEL
LIN {X 0,Y 102.025,Z 461.105,A -85,B 0,C 180,E1 -26548.029,E2 -26548.029} C_VEL
LIN {X 0,Y 105.703,Z 454.2,A -85,B 0,C 180,E1 -26554.391,E2 -26554.391} C_VEL
LIN {X 0,Y 109.501,Z 447.149,A -85,B 0,C 180,E1 -26559.236,E2 -26559.236} C_VEL
LIN {X 0,Y 113.589,Z 439.211,A -85,B 0,C 180,E1 -26563.419,E2 -26563.419} C_VEL
LIN {X 0,Y 118.28,Z 429.452,A -85,B 0,C 180,E1 -26567.286,E2 -26567.286} C_VEL
LIN {X 0,Y 122.861,Z 418.568,A -85,B 0,C 180,E1 -26570.513,E2 -26570.513} C_VEL
LIN {X 0,Y 126.654,Z 408.057,A -85,B 0,C 180,E1 -26572.859,E2 -26572.859} C_VEL
LIN {X 0,Y 130.245,Z 395.609,A -85,B 0,C 180,E1 -26574.936,E2 -26574.936} C_VEL
LIN {X 0,Y 133.235,Z 382.25,A -85,B 0,C 180,E1 -26576.454,E2 -26576.454} C_VEL
LIN {X 0,Y 135.1,Z 369.805,A -85,B 0,C 180,E1 -26577.395,E2 -26577.395} C_VEL
LIN {X 0,Y 138.27,Z 333.542,A -85,B 0,C 180,E1 -26578.969,E2 -26578.969} C_VEL
LIN {X 0,Y 135.474,Z 326.163,A -85,B 0,C 180,E1 -26580.731,E2 -26580.731} C_VEL
LIN {X 0,Y 129.962,Z 315.474,A -85,B 0,C 180,E1 -26584.266,E2 -26584.266} C_VEL
LIN {X 0,Y 124.778,Z 306.612,A -85,B 0,C 180,E1 -26587.972,E2 -26587.972} C_VEL
LIN {X 0,Y 120.044,Z 299.407,A -85,B 0,C 180,E1 -26591.845,E2 -26591.845} C_VEL
LIN {X 0,Y 116.952,Z 295.13,A -85,B 0,C 180,E1 -26594.699,E2 -26594.699} C_VEL
LIN {X 0,Y 114.24,Z 291.332,A -85,B 0,C 180,E1 -26597.542,E2 -26597.542} C_VEL
LIN {X 0,Y 111.141,Z 287.648,A -85,B 0,C 180,E1 -26601.177,E2 -26601.177} C_VEL
LIN {X 0,Y 110.283,Z 285.967,A -85,B 0,C 180,E1 -26602.424,E2 -26602.424} C_VEL
LIN {X 0,Y 107.59,Z 283.83,A -85,B 0,C 180,E1 -26606.29,E2 -26606.29} C_VEL
LIN {X 0,Y 105.837,Z 280.608,A -85,B 0,C 180,E1 -26609.689,E2 -26609.689} C_VEL
LIN {X 0,Y 101.383,Z 275.635,A -85,B 0,C 180,E1 -26627.486,E2 -26627.486} C_VEL
LIN {X 0,Y 101.665,Z 275.97,A -85,B 0,C 180,E1 -26633.564,E2 -26633.564} C_VEL
LIN {X 0,Y 103.169,Z 277.726,A -85,B 0,C 180,E1 -26640.501,E2 -26640.501} C_VEL
LIN {X 0,Y 105.175,Z 279.877,A -85,B 0,C 180,E1 -26645.765,E2 -26645.765} C_VEL
LIN {X 0,Y 106.478,Z 280.805,A -85,B 0,C 180,E1 -26648.243,E2 -26648.243} C_VEL
LIN {X 0,Y 108.232,Z 283.969,A -85,B 0,C 180,E1 -26651.46,E2 -26651.46} C_VEL
LIN {X 0,Y 110.622,Z 286.247,A -85,B 0,C 180,E1 -26654.844,E2 -26654.844} C_VEL
LIN {X 0,Y 112.595,Z 289.454,A -85,B 0,C 180,E1 -26657.449,E2 -26657.449} C_VEL
LIN {X 0,Y 114.391,Z 291.262,A -85,B 0,C 180,E1 -26659.411,E2 -26659.411} C_VEL
LIN {X 0,Y 116.892,Z 294.871,A -85,B 0,C 180,E1 -26662.047,E2 -26662.047} C_VEL
LIN {X 0,Y 118.727,Z 297.497,A -85,B 0,C 180,E1 -26663.797,E2 -26663.797} C_VEL
LIN {X 0,Y 121.677,Z 301.757,A -85,B 0,C 180,E1 -26666.373,E2 -26666.373} C_VEL
LIN {X 0,Y 125.548,Z 307.938,A -85,B 0,C 180,E1 -26669.447,E2 -26669.447} C_VEL
LIN {X 0,Y 130.814,Z 317.287,A -85,B 0,C 180,E1 -26673.152,E2 -26673.152} C_VEL
LIN {X 0,Y 135.089,Z 328.041,A -85,B 0,C 180,E1 -26676.078,E2 -26676.078} C_VEL
LIN {X 0,Y 138.05,Z 336.95,A -85,B 0,C 180,E1 -26678.028,E2 -26678.028} C_VEL
LIN {X 0,Y 134.945,Z 373.646,A -85,B 0,C 180,E1 -26679.703,E2 -26679.703} C_VEL
LIN {X 0,Y 132.598,Z 387.411,A -85,B 0,C 180,E1 -26680.744,E2 -26680.744} C_VEL
LIN {X 0,Y 129.805,Z 399.422,A -85,B 0,C 180,E1 -26682.174,E2 -26682.174} C_VEL
LIN {X 0,Y 126.121,Z 411.354,A -85,B 0,C 180,E1 -26684.152,E2 -26684.152} C_VEL
LIN {X 0,Y 121.888,Z 422.846,A -85,B 0,C 180,E1 -26686.784,E2 -26686.784} C_VEL
LIN {X 0,Y 117.83,Z 432.119,A -85,B 0,C 180,E1 -26689.557,E2 -26689.557} C_VEL
LIN {X 0,Y 113.703,Z 440.973,A -85,B 0,C 180,E1 -26693.048,E2 -26693.048} C_VEL
LIN {X 0,Y 109.731,Z 448.831,A -85,B 0,C 180,E1 -26697.056,E2 -26697.056} C_VEL
LIN {X 0,Y 105.587,Z 456.531,A -85,B 0,C 180,E1 -26702.226,E2 -26702.226} C_VEL
LIN {X 0,Y 102.222,Z 462.738,A -85,B 0,C 180,E1 -26707.778,E2 -26707.778} C_VEL
LIN {X 0,Y 99.898,Z 467.656,A -85,B 0,C 180,E1 -26713.652,E2 -26713.652} C_VEL
LIN {X 0,Y 98.501,Z 471.419,A -85,B 0,C 180,E1 -26719.722,E2 -26719.722} C_VEL
LIN {X 0,Y 97.913,Z 474.134,A -85,B 0,C 180,E1 -26725.881,E2 -26725.881} C_VEL
LIN {X 0,Y 97.962,Z 475.405,A -85,B 0,C 180,E1 -26729.997,E2 -26729.997} C_VEL
LIN {X 0,Y 97.914,Z 476.266,A -85,B 0,C 180,E1 -26734.113,E2 -26734.113} C_VEL
LIN {X 0,Y 98.227,Z 476.708,A -85,B 0,C 180,E1 -26738.224,E2 -26738.224} C_VEL
LIN {X 0,Y 100.088,Z 476.421,A -85,B 0,C 180,E1 -26746.309,E2 -26746.309} C_VEL
LIN {X 0,Y 103.563,Z 474.627,A -85,B 0,C 180,E1 -26754.024,E2 -26754.024} C_VEL
LIN {X 0,Y 109.006,Z 471.18,A -85,B 0,C 180,E1 -26761.046,E2 -26761.046} C_VEL
LIN {X 0,Y 113.948,Z 467.483,A -85,B 0,C 180,E1 -26765.865,E2 -26765.865} C_VEL
LIN {X 0,Y 119.597,Z 462.717,A -85,B 0,C 180,E1 -26770.267,E2 -26770.267} C_VEL
LIN {X 0,Y 127.087,Z 455.63,A -85,B 0,C 180,E1 -26774.832,E2 -26774.832} C_VEL
LIN {X 0,Y 134.162,Z 447.919,A -85,B 0,C 180,E1 -26778.282,E2 -26778.282} C_VEL
LIN {X 0,Y 140.328,Z 440.113,A -85,B 0,C 180,E1 -26780.917,E2 -26780.917} C_VEL
LIN {X 0,Y 146.947,Z 430.619,A -85,B 0,C 180,E1 -26783.231,E2 -26783.231} C_VEL
LIN {X 0,Y 153.026,Z 420.161,A -85,B 0,C 180,E1 -26785.175,E2 -26785.175} C_VEL
LIN {X 0,Y 158.583,Z 408.476,A -85,B 0,C 180,E1 -26786.767,E2 -26786.767} C_VEL
LIN {X 0,Y 163.14,Z 396.139,A -85,B 0,C 180,E1 -26788.004,E2 -26788.004} C_VEL
LIN {X 0,Y 166.848,Z 382.95,A -85,B 0,C 180,E1 -26788.857,E2 -26788.857} C_VEL
LIN {X 0,Y 167.38,Z 380.412,A -85,B 0,C 180,E1 -26788.985,E2 -26788.985} C_VEL
LIN {X 0,Y 167.891,Z 376.625,A -85,B 0,C 180,E1 -26789.369,E2 -26789.369} C_VEL
LIN {X 0,Y 167.791,Z 370.768,A -85,B 0,C 180,E1 -26790.513,E2 -26790.513} C_VEL
LIN {X 0,Y 167.52,Z 364.873,A -85,B 0,C 180,E1 -26791.642,E2 -26791.642} C_VEL
LIN {X 0,Y 167.696,Z 361.02,A -85,B 0,C 180,E1 -26791.996,E2 -26791.996} C_VEL
LIN {X 0,Y 167.607,Z 359.926,A -85,B 0,C 180,E1 -26792.244,E2 -26792.244} C_VEL
LIN {X 0,Y 165.835,Z 354.134,A -85,B 0,C 180,E1 -26795.182,E2 -26795.182} C_VEL
LIN {X 0,Y 164.51,Z 350.897,A -85,B 0,C 180,E1 -26797.648,E2 -26797.648} C_VEL
LIN {X 0,Y 162.862,Z 347.319,A -85,B 0,C 180,E1 -26801.895,E2 -26801.895} C_VEL
LIN {X 0,Y 161.887,Z 345.002,A -85,B 0,C 180,E1 -26808.687,E2 -26808.687} C_VEL
LIN {X 0,Y 162.001,Z 345.31,A -85,B 0,C 180,E1 -26810.8,E2 -26810.8} C_VEL
LIN {X 0,Y 163.073,Z 347.128,A -85,B 0,C 180,E1 -26815.814,E2 -26815.814} C_VEL
LIN {X 0,Y 164.863,Z 351.349,A -85,B 0,C 180,E1 -26820.238,E2 -26820.238} C_VEL
LIN {X 0,Y 166.437,Z 355.012,A -85,B 0,C 180,E1 -26822.95,E2 -26822.95} C_VEL
LIN {X 0,Y 167.905,Z 358.648,A -85,B 0,C 180,E1 -26825.125,E2 -26825.125} C_VEL
LIN {X 0,Y 165.95,Z 373.748,A -85,B 0,C 180,E1 -26825.661,E2 -26825.661} C_VEL
LIN {X 0,Y 163.283,Z 385.734,A -85,B 0,C 180,E1 -26826.241,E2 -26826.241} C_VEL
LIN {X 0,Y 159.681,Z 397.46,A -85,B 0,C 180,E1 -26827.124,E2 -26827.124} C_VEL
LIN {X 0,Y 155.355,Z 408.35,A -85,B 0,C 180,E1 -26828.295,E2 -26828.295} C_VEL
LIN {X 0,Y 149.792,Z 419.457,A -85,B 0,C 180,E1 -26829.857,E2 -26829.857} C_VEL
LIN {X 0,Y 143.57,Z 429.662,A -85,B 0,C 180,E1 -26831.768,E2 -26831.768} C_VEL
LIN {X 0,Y 136.494,Z 439.417,A -85,B 0,C 180,E1 -26834.258,E2 -26834.258} C_VEL
LIN {X 0,Y 128.846,Z 448.212,A -85,B 0,C 180,E1 -26837.351,E2 -26837.351} C_VEL
LIN {X 0,Y 120.731,Z 456.211,A -85,B 0,C 180,E1 -26841.356,E2 -26841.356} C_VEL
LIN {X 0,Y 113.836,Z 462.049,A -85,B 0,C 180,E1 -26845.591,E2 -26845.591} C_VEL
LIN {X 0,Y 106.718,Z 467.212,A -85,B 0,C 180,E1 -26851.122,E2 -26851.122} C_VEL
LIN {X 0,Y 102.861,Z 469.692,A -85,B 0,C 180,E1 -26854.932,E2 -26854.932} C_VEL
LIN {X 0,Y 99.014,Z 471.832,A -85,B 0,C 180,E1 -26859.684,E2 -26859.684} C_VEL
LIN {X 0,Y 96.59,Z 472.976,A -85,B 0,C 180,E1 -26863.319,E2 -26863.319} C_VEL
LIN {X 0,Y 94.05,Z 473.935,A -85,B 0,C 180,E1 -26868.329,E2 -26868.329} C_VEL
LIN {X 0,Y 92.445,Z 474.27,A -85,B 0,C 180,E1 -26872.546,E2 -26872.546} C_VEL
LIN {X 0,Y 91.086,Z 474.177,A -85,B 0,C 180,E1 -26878.043,E2 -26878.043} C_VEL
LIN {X 0,Y 90.447,Z 473.673,A -85,B 0,C 180,E1 -26882.215,E2 -26882.215} C_VEL
LIN {X 0,Y 90.25,Z 472.114,A -85,B 0,C 180,E1 -26889.094,E2 -26889.094} C_VEL
LIN {X 0,Y 91.136,Z 469.228,A -85,B 0,C 180,E1 -26896.628,E2 -26896.628} C_VEL
LIN {X 0,Y 93.007,Z 465.271,A -85,B 0,C 180,E1 -26903.632,E2 -26903.632} C_VEL
LIN {X 0,Y 95.609,Z 460.318,A -85,B 0,C 180,E1 -26910.003,E2 -26910.003} C_VEL
LIN {X 0,Y 98.803,Z 454.743,A -85,B 0,C 180,E1 -26915.399,E2 -26915.399} C_VEL
LIN {X 0,Y 103.039,Z 447.341,A -85,B 0,C 180,E1 -26920.814,E2 -26920.814} C_VEL
LIN {X 0,Y 107.373,Z 439.418,A -85,B 0,C 180,E1 -26925.181,E2 -26925.181} C_VEL
LIN {X 0,Y 112.304,Z 429.696,A -85,B 0,C 180,E1 -26929.184,E2 -26929.184} C_VEL
LIN {X 0,Y 117.107,Z 418.843,A -85,B 0,C 180,E1 -26932.497,E2 -26932.497} C_VEL
LIN {X 0,Y 121.666,Z 406.689,A -85,B 0,C 180,E1 -26935.218,E2 -26935.218} C_VEL
LIN {X 0,Y 125.371,Z 393.945,A -85,B 0,C 180,E1 -26937.278,E2 -26937.278} C_VEL
LIN {X 0,Y 128.373,Z 380.636,A -85,B 0,C 180,E1 -26938.727,E2 -26938.727} C_VEL
LIN {X 0,Y 130.29,Z 367.512,A -85,B 0,C 180,E1 -26939.614,E2 -26939.614} C_VEL
LIN {X 0,Y 133.129,Z 335.635,A -85,B 0,C 180,E1 -26941.007,E2 -26941.007} C_VEL
LIN {X 0,Y 130.841,Z 329.586,A -85,B 0,C 180,E1 -26942.592,E2 -26942.592} C_VEL
LIN {X 0,Y 124.969,Z 318.097,A -85,B 0,C 180,E1 -26946.723,E2 -26946.723} C_VEL
LIN {X 0,Y 119.393,Z 308.563,A -85,B 0,C 180,E1 -26951.28,E2 -26951.28} C_VEL
LIN {X 0,Y 114.522,Z 301.323,A -85,B 0,C 180,E1 -26955.934,E2 -26955.934} C_VEL
LIN {X 0,Y 111.346,Z 296.932,A -85,B 0,C 180,E1 -26959.529,E2 -26959.529} C_VEL
LIN {X 0,Y 108.781,Z 293.435,A -85,B 0,C 180,E1 -26962.932,E2 -26962.932} C_VEL
LIN {X 0,Y 108.118,Z 292.375,A -85,B 0,C 180,E1 -26963.939,E2 -26963.939} C_VEL
LIN {X 0,Y 105.649,Z 290.045,A -85,B 0,C 180,E1 -26967.864,E2 -26967.864} C_VEL
LIN {X 0,Y 104.313,Z 287.29,A -85,B 0,C 180,E1 -26970.775,E2 -26970.775} C_VEL
LIN {X 0,Y 100.962,Z 284.558,A -85,B 0,C 180,E1 -26980.707,E2 -26980.707} C_VEL
LIN {X 0,Y 100.401,Z 282.624,A -85,B 0,C 180,E1 -26987.892,E2 -26987.892} C_VEL
LIN {X 0,Y 100.681,Z 283.035,A -85,B 0,C 180,E1 -26993.501,E2 -26993.501} C_VEL
LIN {X 0,Y 102.053,Z 284.765,A -85,B 0,C 180,E1 -27000.013,E2 -27000.013} C_VEL
LIN {X 0,Y 104.233,Z 286.96,A -85,B 0,C 180,E1 -27005.818,E2 -27005.818} C_VEL
LIN {X 0,Y 104.878,Z 287.459,A -85,B 0,C 180,E1 -27007.11,E2 -27007.11} C_VEL
LIN {X 0,Y 106.382,Z 290.356,A -85,B 0,C 180,E1 -27010.119,E2 -27010.119} C_VEL
LIN {X 0,Y 108.66,Z 292.829,A -85,B 0,C 180,E1 -27013.641,E2 -27013.641} C_VEL
LIN {X 0,Y 110.886,Z 296.224,A -85,B 0,C 180,E1 -27016.717,E2 -27016.717} C_VEL
LIN {X 0,Y 112.197,Z 297.758,A -85,B 0,C 180,E1 -27018.264,E2 -27018.264} C_VEL
LIN {X 0,Y 115.395,Z 302.467,A -85,B 0,C 180,E1 -27021.783,E2 -27021.783} C_VEL
LIN {X 0,Y 118.733,Z 307.482,A -85,B 0,C 180,E1 -27024.956,E2 -27024.956} C_VEL
LIN {X 0,Y 123.221,Z 315.038,A -85,B 0,C 180,E1 -27028.761,E2 -27028.761} C_VEL
LIN {X 0,Y 127.328,Z 322.975,A -85,B 0,C 180,E1 -27031.869,E2 -27031.869} C_VEL
LIN {X 0,Y 131.433,Z 334.112,A -85,B 0,C 180,E1 -27034.909,E2 -27034.909} C_VEL
LIN {X 0,Y 132.878,Z 338.788,A -85,B 0,C 180,E1 -27035.967,E2 -27035.967} C_VEL
LIN {X 0,Y 129.712,Z 374.237,A -85,B 0,C 180,E1 -27037.623,E2 -27037.623} C_VEL
LIN {X 0,Y 127.329,Z 387.532,A -85,B 0,C 180,E1 -27038.644,E2 -27038.644} C_VEL
LIN {X 0,Y 124.52,Z 399.156,A -85,B 0,C 180,E1 -27040.047,E2 -27040.047} C_VEL
LIN {X 0,Y 120.667,Z 411.131,A -85,B 0,C 180,E1 -27042.043,E2 -27042.043} C_VEL
LIN {X 0,Y 116.237,Z 422.649,A -85,B 0,C 180,E1 -27044.726,E2 -27044.726} C_VEL
LIN {X 0,Y 111.978,Z 431.94,A -85,B 0,C 180,E1 -27047.566,E2 -27047.566} C_VEL
LIN {X 0,Y 107.063,Z 441.847,A -85,B 0,C 180,E1 -27051.656,E2 -27051.656} C_VEL
LIN {X 0,Y 102.926,Z 449.556,A -85,B 0,C 180,E1 -27055.899,E2 -27055.899} C_VEL
LIN {X 0,Y 98.667,Z 456.957,A -85,B 0,C 180,E1 -27061.259,E2 -27061.259} C_VEL
LIN {X 0,Y 94.638,Z 463.975,A -85,B 0,C 180,E1 -27068.2,E2 -27068.2} C_VEL
LIN {X 0,Y 92.442,Z 468.605,A -85,B 0,C 180,E1 -27074.565,E2 -27074.565} C_VEL
LIN {X 0,Y 91.179,Z 472.1,A -85,B 0,C 180,E1 -27081.128,E2 -27081.128} C_VEL
LIN {X 0,Y 90.828,Z 473.839,A -85,B 0,C 180,E1 -27085.559,E2 -27085.559} C_VEL
LIN {X 0,Y 90.861,Z 475.155,A -85,B 0,C 180,E1 -27089.996,E2 -27089.996} C_VEL
LIN {X 0,Y 90.829,Z 476.059,A -85,B 0,C 180,E1 -27094.434,E2 -27094.434} C_VEL
LIN {X 0,Y 91.192,Z 476.576,A -85,B 0,C 180,E1 -27098.863,E2 -27098.863} C_VEL
LIN {X 0,Y 93.277,Z 476.389,A -85,B 0,C 180,E1 -27107.537,E2 -27107.537} C_VEL
LIN {X 0,Y 97.103,Z 474.702,A -85,B 0,C 180,E1 -27115.734,E2 -27115.734} C_VEL
LIN {X 0,Y 99.833,Z 473.267,A -85,B 0,C 180,E1 -27119.52,E2 -27119.52} C_VEL
LIN {X 0,Y 104.678,Z 470.327,A -85,B 0,C 180,E1 -27124.794,E2 -27124.794} C_VEL
LIN {X 0,Y 110.223,Z 466.385,A -85,B 0,C 180,E1 -27129.61,E2 -27129.61} C_VEL
LIN {X 0,Y 116.441,Z 461.353,A -85,B 0,C 180,E1 -27133.951,E2 -27133.951} C_VEL
LIN {X 0,Y 123.383,Z 455.072,A -85,B 0,C 180,E1 -27137.769,E2 -27137.769} C_VEL
LIN {X 0,Y 130.884,Z 447.259,A -85,B 0,C 180,E1 -27141.128,E2 -27141.128} C_VEL
LIN {X 0,Y 135.999,Z 441.107,A -85,B 0,C 180,E1 -27143.22,E2 -27143.22} C_VEL
LIN {X 0,Y 143.554,Z 430.794,A -85,B 0,C 180,E1 -27145.701,E2 -27145.701} C_VEL
LIN {X 0,Y 149.851,Z 420.389,A -85,B 0,C 180,E1 -27147.581,E2 -27147.581} C_VEL
LIN {X 0,Y 155.589,Z 408.821,A -85,B 0,C 180,E1 -27149.114,E2 -27149.114} C_VEL
LIN {X 0,Y 160.294,Z 396.597,A -85,B 0,C 180,E1 -27150.299,E2 -27150.299} C_VEL
LIN {X 0,Y 164.112,Z 383.565,A -85,B 0,C 180,E1 -27151.118,E2 -27151.118} C_VEL
LIN {X 0,Y 166.637,Z 370.152,A -85,B 0,C 180,E1 -27151.689,E2 -27151.689} C_VEL
LIN {X 0,Y 167.696,Z 361.02,A -85,B 0,C 180,E1 -27151.996,E2 -27151.996} C_VEL
LIN {X 0,Y 167.615,Z 359.12,A -85,B 0,C 180,E1 -27152.353,E2 -27152.353} C_VEL
LIN {X 0,Y 167.017,Z 357.683,A -85,B 0,C 180,E1 -27153.21,E2 -27153.21} C_VEL
LIN {X 0,Y 165.826,Z 357.059,A -85,B 0,C 180,E1 -27154.694,E2 -27154.694} C_VEL
LIN {X 0,Y 163.276,Z 357.451,A -85,B 0,C 180,E1 -27158.24,E2 -27158.24} C_VEL
LIN {X 0,Y 162.868,Z 357.05,A -85,B 0,C 180,E1 -27159.06,E2 -27159.06} C_VEL
LIN {X 0,Y 161.789,Z 354.229,A -85,B 0,C 180,E1 -27162.289,E2 -27162.289} C_VEL
LIN {X 0,Y 160.954,Z 352.049,A -85,B 0,C 180,E1 -27168.62,E2 -27168.62} C_VEL
LIN {X 0,Y 161.051,Z 352.42,A -85,B 0,C 180,E1 -27170.745,E2 -27170.745} C_VEL
LIN {X 0,Y 161.915,Z 353.965,A -85,B 0,C 180,E1 -27175.207,E2 -27175.207} C_VEL
LIN {X 0,Y 163.517,Z 358.063,A -85,B 0,C 180,E1 -27179.558,E2 -27179.558} C_VEL
LIN {X 0,Y 165.227,Z 362.519,A -85,B 0,C 180,E1 -27182.74,E2 -27182.74} C_VEL
LIN {X 0,Y 165.351,Z 363.008,A -85,B 0,C 180,E1 -27182.97,E2 -27182.97} C_VEL
LIN {X 0,Y 163.162,Z 377.038,A -85,B 0,C 180,E1 -27183.433,E2 -27183.433} C_VEL
LIN {X 0,Y 160.381,Z 388.206,A -85,B 0,C 180,E1 -27184.02,E2 -27184.02} C_VEL
LIN {X 0,Y 156.557,Z 399.529,A -85,B 0,C 180,E1 -27184.875,E2 -27184.875} C_VEL
LIN {X 0,Y 151.114,Z 412.033,A -85,B 0,C 180,E1 -27186.247,E2 -27186.247} C_VEL
LIN {X 0,Y 145.391,Z 422.419,A -85,B 0,C 180,E1 -27187.748,E2 -27187.748} C_VEL
LIN {X 0,Y 138.208,Z 433.105,A -85,B 0,C 180,E1 -27189.874,E2 -27189.874} C_VEL
LIN {X 0,Y 130.763,Z 442.391,A -85,B 0,C 180,E1 -27192.403,E2 -27192.403} C_VEL
LIN {X 0,Y 123.769,Z 449.804,A -85,B 0,C 180,E1 -27195.147,E2 -27195.147} C_VEL
LIN {X 0,Y 116.7,Z 456.32,A -85,B 0,C 180,E1 -27198.476,E2 -27198.476} C_VEL
LIN {X 0,Y 109.332,Z 462.162,A -85,B 0,C 180,E1 -27202.672,E2 -27202.672} C_VEL
LIN {X 0,Y 102.826,Z 466.619,A -85,B 0,C 180,E1 -27207.319,E2 -27207.319} C_VEL
LIN {X 0,Y 96.51,Z 470.285,A -85,B 0,C 180,E1 -27213.136,E2 -27213.136} C_VEL
LIN {X 0,Y 91.324,Z 472.76,A -85,B 0,C 180,E1 -27219.691,E2 -27219.691} C_VEL
LIN {X 0,Y 87.64,Z 474.038,A -85,B 0,C 180,E1 -27226.172,E2 -27226.172} C_VEL
LIN {X 0,Y 84.679,Z 474.365,A -85,B 0,C 180,E1 -27234.486,E2 -27234.486} C_VEL
LIN {X 0,Y 83.646,Z 473.957,A -85,B 0,C 180,E1 -27239.732,E2 -27239.732} C_VEL
LIN {X 0,Y 83.122,Z 472.264,A -85,B 0,C 180,E1 -27248.393,E2 -27248.393} C_VEL
LIN {X 0,Y 84.272,Z 468.778,A -85,B 0,C 180,E1 -27257.97,E2 -27257.97} C_VEL
LIN {X 0,Y 86.325,Z 464.745,A -85,B 0,C 180,E1 -27265.334,E2 -27265.334} C_VEL
LIN {X 0,Y 89.329,Z 459.51,A -85,B 0,C 180,E1 -27272.258,E2 -27272.258} C_VEL
LIN {X 0,Y 93.44,Z 452.868,A -85,B 0,C 180,E1 -27278.655,E2 -27278.655} C_VEL
LIN {X 0,Y 98.418,Z 444.523,A -85,B 0,C 180,E1 -27284.477,E2 -27284.477} C_VEL
LIN {X 0,Y 103.271,Z 435.963,A -85,B 0,C 180,E1 -27288.863,E2 -27288.863} C_VEL
LIN {X 0,Y 108.115,Z 426.555,A -85,B 0,C 180,E1 -27292.47,E2 -27292.47} C_VEL
LIN {X 0,Y 112.705,Z 416.342,A -85,B 0,C 180,E1 -27295.389,E2 -27295.389} C_VEL
LIN {X 0,Y 116.903,Z 405.175,A -85,B 0,C 180,E1 -27297.772,E2 -27297.772} C_VEL
LIN {X 0,Y 120.534,Z 392.917,A -85,B 0,C 180,E1 -27299.715,E2 -27299.715} C_VEL
LIN {X 0,Y 123.429,Z 380.325,A -85,B 0,C 180,E1 -27301.05,E2 -27301.05} C_VEL
LIN {X 0,Y 125.482,Z 366.42,A -85,B 0,C 180,E1 -27301.964,E2 -27301.964} C_VEL
LIN {X 0,Y 128.05,Z 337.344,A -85,B 0,C 180,E1 -27303.291,E2 -27303.291} C_VEL
LIN {X 0,Y 125.152,Z 330.666,A -85,B 0,C 180,E1 -27305.415,E2 -27305.415} C_VEL
LIN {X 0,Y 120.082,Z 320.626,A -85,B 0,C 180,E1 -27309.485,E2 -27309.485} C_VEL
LIN {X 0,Y 115.742,Z 313.248,A -85,B 0,C 180,E1 -27313.416,E2 -27313.416} C_VEL
LIN {X 0,Y 112.142,Z 307.478,A -85,B 0,C 180,E1 -27317.235,E2 -27317.235} C_VEL
LIN {X 0,Y 109.035,Z 303.07,A -85,B 0,C 180,E1 -27321.026,E2 -27321.026} C_VEL
LIN {X 0,Y 106.173,Z 298.918,A -85,B 0,C 180,E1 -27325.275,E2 -27325.275} C_VEL
LIN {X 0,Y 103.767,Z 296.188,A -85,B 0,C 180,E1 -27329.556,E2 -27329.556} C_VEL
LIN {X 0,Y 102.773,Z 294.088,A -85,B 0,C 180,E1 -27331.973,E2 -27331.973} C_VEL
LIN {X 0,Y 99.46,Z 289.742,A -85,B 0,C 180,E1 -27347.776,E2 -27347.776} C_VEL
LIN {X 0,Y 99.66,Z 289.943,A -85,B 0,C 180,E1 -27352.671,E2 -27352.671} C_VEL
LIN {X 0,Y 100.882,Z 291.648,A -85,B 0,C 180,E1 -27359.265,E2 -27359.265} C_VEL
LIN {X 0,Y 103.333,Z 294.324,A -85,B 0,C 180,E1 -27366.022,E2 -27366.022} C_VEL
LIN {X 0,Y 105.322,Z 297.711,A -85,B 0,C 180,E1 -27370.085,E2 -27370.085} C_VEL
LIN {X 0,Y 106.73,Z 299.354,A -85,B 0,C 180,E1 -27372.39,E2 -27372.39} C_VEL
LIN {X 0,Y 109.098,Z 302.919,A -85,B 0,C 180,E1 -27375.842,E2 -27375.842} C_VEL
LIN {X 0,Y 110.207,Z 304.531,A -85,B 0,C 180,E1 -27377.276,E2 -27377.276} C_VEL
LIN {X 0,Y 113.134,Z 308.967,A -85,B 0,C 180,E1 -27380.702,E2 -27380.702} C_VEL
LIN {X 0,Y 116.831,Z 314.8,A -85,B 0,C 180,E1 -27384.422,E2 -27384.422} C_VEL
LIN {X 0,Y 122.08,Z 324.611,A -85,B 0,C 180,E1 -27389.036,E2 -27389.036} C_VEL
LIN {X 0,Y 124.517,Z 330.476,A -85,B 0,C 180,E1 -27391.041,E2 -27391.041} C_VEL
LIN {X 0,Y 127.912,Z 340.643,A -85,B 0,C 180,E1 -27393.757,E2 -27393.757} C_VEL
LIN {X 0,Y 124.809,Z 373.872,A -85,B 0,C 180,E1 -27395.315,E2 -27395.315} C_VEL
LIN {X 0,Y 122.395,Z 387.027,A -85,B 0,C 180,E1 -27396.317,E2 -27396.317} C_VEL
LIN {X 0,Y 119.421,Z 398.875,A -85,B 0,C 180,E1 -27397.735,E2 -27397.735} C_VEL
LIN {X 0,Y 115.395,Z 410.898,A -85,B 0,C 180,E1 -27399.74,E2 -27399.74} C_VEL
LIN {X 0,Y 110.751,Z 422.439,A -85,B 0,C 180,E1 -27402.46,E2 -27402.46} C_VEL
LIN {X 0,Y 106.277,Z 431.747,A -85,B 0,C 180,E1 -27405.358,E2 -27405.358} C_VEL
LIN {X 0,Y 101.757,Z 440.45,A -85,B 0,C 180,E1 -27408.991,E2 -27408.991} C_VEL
LIN {X 0,Y 97.269,Z 448.281,A -85,B 0,C 180,E1 -27413.263,E2 -27413.263} C_VEL
LIN {X 0,Y 92.45,Z 456.239,A -85,B 0,C 180,E1 -27419.124,E2 -27419.124} C_VEL
LIN {X 0,Y 89.192,Z 461.547,A -85,B 0,C 180,E1 -27424.314,E2 -27424.314} C_VEL
LIN {X 0,Y 86.303,Z 466.676,A -85,B 0,C 180,E1 -27430.986,E2 -27430.986} C_VEL
LIN {X 0,Y 84.545,Z 470.637,A -85,B 0,C 180,E1 -27438.002,E2 -27438.002} C_VEL
LIN {X 0,Y 83.763,Z 473.536,A -85,B 0,C 180,E1 -27445.183,E2 -27445.183} C_VEL
LIN {X 0,Y 83.783,Z 474.897,A -85,B 0,C 180,E1 -27449.996,E2 -27449.996} C_VEL
LIN {X 0,Y 83.764,Z 475.845,A -85,B 0,C 180,E1 -27454.809,E2 -27454.809} C_VEL
LIN {X 0,Y 85.094,Z 476.593,A -85,B 0,C 180,E1 -27464.342,E2 -27464.342} C_VEL
LIN {X 0,Y 88.365,Z 475.751,A -85,B 0,C 180,E1 -27473.428,E2 -27473.428} C_VEL
LIN {X 0,Y 93.711,Z 473.402,A -85,B 0,C 180,E1 -27481.662,E2 -27481.662} C_VEL
LIN {X 0,Y 98.922,Z 470.548,A -85,B 0,C 180,E1 -27487.144,E2 -27487.144} C_VEL
LIN {X 0,Y 106.316,Z 465.72,A -85,B 0,C 180,E1 -27493.111,E2 -27493.111} C_VEL
LIN {X 0,Y 113.83,Z 459.917,A -85,B 0,C 180,E1 -27497.803,E2 -27497.803} C_VEL
LIN {X 0,Y 121.271,Z 453.323,A -85,B 0,C 180,E1 -27501.472,E2 -27501.472} C_VEL
LIN {X 0,Y 129.219,Z 445.174,A -85,B 0,C 180,E1 -27504.664,E2 -27504.664} C_VEL
LIN {X 0,Y 136.123,Z 436.863,A -85,B 0,C 180,E1 -27507.027,E2 -27507.027} C_VEL
LIN {X 0,Y 143.297,Z 426.657,A -85,B 0,C 180,E1 -27509.119,E2 -27509.119} C_VEL
LIN {X 0,Y 149.899,Z 415.27,A -85,B 0,C 180,E1 -27510.831,E2 -27510.831} C_VEL
LIN {X 0,Y 155.117,Z 404.096,A -85,B 0,C 180,E1 -27512.062,E2 -27512.062} C_VEL
LIN {X 0,Y 159.125,Z 393.125,A -85,B 0,C 180,E1 -27512.961,E2 -27512.961} C_VEL
LIN {X 0,Y 162.863,Z 379.215,A -85,B 0,C 180,E1 -27513.684,E2 -27513.684} C_VEL
LIN {X 0,Y 164.957,Z 366.585,A -85,B 0,C 180,E1 -27514.156,E2 -27514.156} C_VEL
LIN {X 0,Y 165.209,Z 364.05,A -85,B 0,C 180,E1 -27514.276,E2 -27514.276} C_VEL
LIN {X 0,Y 163.912,Z 359.457,A -85,B 0,C 180,E1 -27516.793,E2 -27516.793} C_VEL
LIN {X 0,Y 162.868,Z 357.05,A -85,B 0,C 180,E1 -27519.06,E2 -27519.06} C_VEL
LIN {X 0,Y 162.228,Z 356.755,A -85,B 0,C 180,E1 -27520.432,E2 -27520.432} C_VEL
LIN {X 0,Y 161.142,Z 358.136,A -85,B 0,C 180,E1 -27522.726,E2 -27522.726} C_VEL
LIN {X 0,Y 160.312,Z 359.744,A -85,B 0,C 180,E1 -27525.06,E2 -27525.06} C_VEL
LIN {X 0,Y 160.077,Z 359.779,A -85,B 0,C 180,E1 -27526.495,E2 -27526.495} C_VEL
LIN {X 0,Y 160.016,Z 359.141,A -85,B 0,C 180,E1 -27528.553,E2 -27528.553} C_VEL
LIN {X 0,Y 160.082,Z 359.335,A -85,B 0,C 180,E1 -27530.283,E2 -27530.283} C_VEL
LIN {X 0,Y 160.831,Z 361.002,A -85,B 0,C 180,E1 -27534.821,E2 -27534.821} C_VEL
LIN {X 0,Y 162.183,Z 364.731,A -85,B 0,C 180,E1 -27538.824,E2 -27538.824} C_VEL
LIN {X 0,Y 162.972,Z 367.205,A -85,B 0,C 180,E1 -27540.691,E2 -27540.691} C_VEL
LIN {X 0,Y 160.311,Z 381.252,A -85,B 0,C 180,E1 -27541.166,E2 -27541.166} C_VEL
LIN {X 0,Y 156.384,Z 394.499,A -85,B 0,C 180,E1 -27541.964,E2 -27541.964} C_VEL
LIN {X 0,Y 151.647,Z 406.363,A -85,B 0,C 180,E1 -27543.016,E2 -27543.016} C_VEL
LIN {X 0,Y 146.232,Z 417.045,A -85,B 0,C 180,E1 -27544.28,E2 -27544.28} C_VEL
LIN {X 0,Y 139.71,Z 427.491,A -85,B 0,C 180,E1 -27545.935,E2 -27545.935} C_VEL
LIN {X 0,Y 133.009,Z 436.424,A -85,B 0,C 180,E1 -27547.833,E2 -27547.833} C_VEL
LIN {X 0,Y 125.05,Z 445.363,A -85,B 0,C 180,E1 -27550.432,E2 -27550.432} C_VEL
LIN {X 0,Y 117.24,Z 452.807,A -85,B 0,C 180,E1 -27553.458,E2 -27553.458} C_VEL
LIN {X 0,Y 108.73,Z 459.715,A -85,B 0,C 180,E1 -27557.512,E2 -27557.512} C_VEL
LIN {X 0,Y 101.968,Z 464.402,A -85,B 0,C 180,E1 -27561.503,E2 -27561.503} C_VEL
LIN {X 0,Y 94.606,Z 468.707,A -85,B 0,C 180,E1 -27566.954,E2 -27566.954} C_VEL
LIN {X 0,Y 87.613,Z 472.053,A -85,B 0,C 180,E1 -27574.14,E2 -27574.14} C_VEL
LIN {X 0,Y 81.413,Z 474.139,A -85,B 0,C 180,E1 -27583.653,E2 -27583.653} C_VEL
LIN {X 0,Y 78.394,Z 474.52,A -85,B 0,C 180,E1 -27591.137,E2 -27591.137} C_VEL
LIN {X 0,Y 76.99,Z 474.201,A -85,B 0,C 180,E1 -27596.796,E2 -27596.796} C_VEL
LIN {X 0,Y 76.195,Z 473.446,A -85,B 0,C 180,E1 -27602.542,E2 -27602.542} C_VEL
LIN {X 0,Y 76.029,Z 472.212,A -85,B 0,C 180,E1 -27608.304,E2 -27608.304} C_VEL
LIN {X 0,Y 76.858,Z 469.469,A -85,B 0,C 180,E1 -27616.79,E2 -27616.79} C_VEL
LIN {X 0,Y 78.9,Z 465.616,A -85,B 0,C 180,E1 -27624.894,E2 -27624.894} C_VEL
LIN {X 0,Y 81.944,Z 460.58,A -85,B 0,C 180,E1 -27632.462,E2 -27632.462} C_VEL
LIN {X 0,Y 86.147,Z 454.189,A -85,B 0,C 180,E1 -27639.394,E2 -27639.394} C_VEL
LIN {X 0,Y 91.32,Z 446.2,A -85,B 0,C 180,E1 -27645.63,E2 -27645.63} C_VEL
LIN {X 0,Y 96.363,Z 437.946,A -85,B 0,C 180,E1 -27650.273,E2 -27650.273} C_VEL
LIN {X 0,Y 101.925,Z 427.843,A -85,B 0,C 180,E1 -27654.442,E2 -27654.442} C_VEL
LIN {X 0,Y 106.725,Z 417.898,A -85,B 0,C 180,E1 -27657.452,E2 -27657.452} C_VEL
LIN {X 0,Y 111.104,Z 407.155,A -85,B 0,C 180,E1 -27659.88,E2 -27659.88} C_VEL
LIN {X 0,Y 115.233,Z 394.254,A -85,B 0,C 180,E1 -27661.998,E2 -27661.998} C_VEL
LIN {X 0,Y 118.413,Z 381.294,A -85,B 0,C 180,E1 -27663.43,E2 -27663.43} C_VEL
LIN {X 0,Y 120.541,Z 368.011,A -85,B 0,C 180,E1 -27664.342,E2 -27664.342} C_VEL
LIN {X 0,Y 123.267,Z 339.745,A -85,B 0,C 180,E1 -27665.597,E2 -27665.597} C_VEL
LIN {X 0,Y 118.856,Z 330.085,A -85,B 0,C 180,E1 -27669.275,E2 -27669.275} C_VEL
LIN {X 0,Y 114.553,Z 321.81,A -85,B 0,C 180,E1 -27673.294,E2 -27673.294} C_VEL
LIN {X 0,Y 111.074,Z 315.885,A -85,B 0,C 180,E1 -27677.045,E2 -27677.045} C_VEL
LIN {X 0,Y 108.935,Z 312.504,A -85,B 0,C 180,E1 -27679.646,E2 -27679.646} C_VEL
LIN {X 0,Y 106.777,Z 309.202,A -85,B 0,C 180,E1 -27682.591,E2 -27682.591} C_VEL
LIN {X 0,Y 104.362,Z 305.417,A -85,B 0,C 180,E1 -27686.556,E2 -27686.556} C_VEL
LIN {X 0,Y 102.145,Z 302.695,A -85,B 0,C 180,E1 -27690.878,E2 -27690.878} C_VEL
LIN {X 0,Y 101.267,Z 300.846,A -85,B 0,C 180,E1 -27693.214,E2 -27693.214} C_VEL
LIN {X 0,Y 98.52,Z 296.866,A -85,B 0,C 180,E1 -27707.657,E2 -27707.657} C_VEL
LIN {X 0,Y 98.748,Z 297.083,A -85,B 0,C 180,E1 -27712.945,E2 -27712.945} C_VEL
LIN {X 0,Y 99.749,Z 298.619,A -85,B 0,C 180,E1 -27718.626,E2 -27718.626} C_VEL
LIN {X 0,Y 101.836,Z 301.081,A -85,B 0,C 180,E1 -27724.9,E2 -27724.9} C_VEL
LIN {X 0,Y 103.928,Z 304.611,A -85,B 0,C 180,E1 -27729.439,E2 -27729.439} C_VEL
LIN {X 0,Y 104.885,Z 305.941,A -85,B 0,C 180,E1 -27731.15,E2 -27731.15} C_VEL
LIN {X 0,Y 108.025,Z 310.827,A -85,B 0,C 180,E1 -27735.943,E2 -27735.943} C_VEL
LIN {X 0,Y 110.815,Z 315.316,A -85,B 0,C 180,E1 -27739.461,E2 -27739.461} C_VEL
LIN {X 0,Y 114.12,Z 320.852,A -85,B 0,C 180,E1 -27743.072,E2 -27743.072} C_VEL
LIN {X 0,Y 119.029,Z 330.558,A -85,B 0,C 180,E1 -27747.721,E2 -27747.721} C_VEL
LIN {X 0,Y 122.199,Z 339.696,A -85,B 0,C 180,E1 -27750.616,E2 -27750.616} C_VEL
LIN {X 0,Y 123.101,Z 342.747,A -85,B 0,C 180,E1 -27751.424,E2 -27751.424} C_VEL
LIN {X 0,Y 119.994,Z 373.941,A -85,B 0,C 180,E1 -27752.873,E2 -27752.873} C_VEL
LIN {X 0,Y 117.465,Z 387.181,A -85,B 0,C 180,E1 -27753.882,E2 -27753.882} C_VEL
LIN {X 0,Y 114.194,Z 399.484,A -85,B 0,C 180,E1 -27755.363,E2 -27755.363} C_VEL
LIN {X 0,Y 109.729,Z 412.128,A -85,B 0,C 180,E1 -27757.566,E2 -27757.566} C_VEL
LIN {X 0,Y 104.815,Z 423.405,A -85,B 0,C 180,E1 -27760.292,E2 -27760.292} C_VEL
LIN {X 0,Y 99.646,Z 433.572,A -85,B 0,C 180,E1 -27763.699,E2 -27763.699} C_VEL
LIN {X 0,Y 94.426,Z 442.757,A -85,B 0,C 180,E1 -27767.94,E2 -27767.94} C_VEL
LIN {X 0,Y 90.646,Z 448.959,A -85,B 0,C 180,E1 -27771.661,E2 -27771.661} C_VEL
LIN {X 0,Y 85.644,Z 456.612,A -85,B 0,C 180,E1 -27777.761,E2 -27777.761} C_VEL
LIN {X 0,Y 81.566,Z 462.743,A -85,B 0,C 180,E1 -27784.476,E2 -27784.476} C_VEL
LIN {X 0,Y 78.793,Z 467.596,A -85,B 0,C 180,E1 -27791.805,E2 -27791.805} C_VEL
LIN {X 0,Y 77.189,Z 471.296,A -85,B 0,C 180,E1 -27799.504,E2 -27799.504} C_VEL
LIN {X 0,Y 76.678,Z 473.193,A -85,B 0,C 180,E1 -27804.737,E2 -27804.737} C_VEL
LIN {X 0,Y 76.694,Z 474.634,A -85,B 0,C 180,E1 -27809.996,E2 -27809.996} C_VEL
LIN {X 0,Y 77.198,Z 476.241,A -85,B 0,C 180,E1 -27820.486,E2 -27820.486} C_VEL
LIN {X 0,Y 79.79,Z 476.329,A -85,B 0,C 180,E1 -27830.625,E2 -27830.625} C_VEL
LIN {X 0,Y 84.517,Z 474.841,A -85,B 0,C 180,E1 -27839.925,E2 -27839.925} C_VEL
LIN {X 0,Y 91.396,Z 471.828,A -85,B 0,C 180,E1 -27847.959,E2 -27847.959} C_VEL
LIN {X 0,Y 97.5,Z 468.44,A -85,B 0,C 180,E1 -27853.213,E2 -27853.213} C_VEL
LIN {X 0,Y 104.3,Z 464.027,A -85,B 0,C 180,E1 -27857.829,E2 -27857.829} C_VEL
LIN {X 0,Y 113.062,Z 457.394,A -85,B 0,C 180,E1 -27862.419,E2 -27862.419} C_VEL
LIN {X 0,Y 121.145,Z 450.218,A -85,B 0,C 180,E1 -27865.754,E2 -27865.754} C_VEL
LIN {X 0,Y 128.066,Z 442.992,A -85,B 0,C 180,E1 -27868.272,E2 -27868.272} C_VEL
LIN {X 0,Y 135.384,Z 434.235,A -85,B 0,C 180,E1 -27870.397,E2 -27870.397} C_VEL
LIN {X 0,Y 142.84,Z 423.52,A -85,B 0,C 180,E1 -27872.324,E2 -27872.324} C_VEL
LIN {X 0,Y 148.922,Z 412.766,A -85,B 0,C 180,E1 -27873.716,E2 -27873.716} C_VEL
LIN {X 0,Y 154.266,Z 400.879,A -85,B 0,C 180,E1 -27874.879,E2 -27874.879} C_VEL
LIN {X 0,Y 158.541,Z 388.615,A -85,B 0,C 180,E1 -27875.671,E2 -27875.671} C_VEL
LIN {X 0,Y 161.713,Z 375.534,A -85,B 0,C 180,E1 -27876.233,E2 -27876.233} C_VEL
LIN {X 0,Y 162.89,Z 367.831,A -85,B 0,C 180,E1 -27876.571,E2 -27876.571} C_VEL
LIN {X 0,Y 162.243,Z 365.42,A -85,B 0,C 180,E1 -27878.155,E2 -27878.155} C_VEL
LIN {X 0,Y 161.53,Z 363.603,A -85,B 0,C 180,E1 -27879.954,E2 -27879.954} C_VEL
LIN {X 0,Y 160.62,Z 361.013,A -85,B 0,C 180,E1 -27883.059,E2 -27883.059} C_VEL
LIN {X 0,Y 160.077,Z 359.779,A -85,B 0,C 180,E1 -27886.495,E2 -27886.495} C_VEL
LIN {X 0,Y 159.953,Z 359.95,A -85,B 0,C 180,E1 -27887.657,E2 -27887.657} C_VEL
LIN {X 0,Y 159.71,Z 361.649,A -85,B 0,C 180,E1 -27889.207,E2 -27889.207} C_VEL
LIN {X 0,Y 159.411,Z 366.416,A -85,B 0,C 180,E1 -27892.203,E2 -27892.203} C_VEL
LIN {X 0,Y 159.557,Z 367.497,A -85,B 0,C 180,E1 -27893.614,E2 -27893.614} C_VEL
LIN {X 0,Y 160.661,Z 371.132,A -85,B 0,C 180,E1 -27897.886,E2 -27897.886} C_VEL
LIN {X 0,Y 160.79,Z 371.657,A -85,B 0,C 180,E1 -27898.337,E2 -27898.337} C_VEL
LIN {X 0,Y 157.735,Z 385.104,A -85,B 0,C 180,E1 -27898.862,E2 -27898.862} C_VEL
LIN {X 0,Y 153.655,Z 397.488,A -85,B 0,C 180,E1 -27899.615,E2 -27899.615} C_VEL
LIN {X 0,Y 148.178,Z 409.863,A -85,B 0,C 180,E1 -27900.745,E2 -27900.745} C_VEL
LIN {X 0,Y 141.534,Z 421.591,A -85,B 0,C 180,E1 -27902.177,E2 -27902.177} C_VEL
LIN {X 0,Y 135.166,Z 430.81,A -85,B 0,C 180,E1 -27903.703,E2 -27903.703} C_VEL
LIN {X 0,Y 128.827,Z 438.59,A -85,B 0,C 180,E1 -27905.406,E2 -27905.406} C_VEL
LIN {X 0,Y 120.613,Z 447.16,A -85,B 0,C 180,E1 -27907.899,E2 -27907.899} C_VEL
LIN {X 0,Y 112.812,Z 454.049,A -85,B 0,C 180,E1 -27910.759,E2 -27910.759} C_VEL
LIN {X 0,Y 105.096,Z 459.876,A -85,B 0,C 180,E1 -27914.167,E2 -27914.167} C_VEL
LIN {X 0,Y 96.557,Z 465.305,A -85,B 0,C 180,E1 -27918.889,E2 -27918.889} C_VEL
LIN {X 0,Y 88.66,Z 469.451,A -85,B 0,C 180,E1 -27924.564,E2 -27924.564} C_VEL
LIN {X 0,Y 82.042,Z 472.263,A -85,B 0,C 180,E1 -27931.068,E2 -27931.068} C_VEL
LIN {X 0,Y 78.214,Z 473.555,A -85,B 0,C 180,E1 -27936.038,E2 -27936.038} C_VEL
LIN {X 0,Y 74.986,Z 474.308,A -85,B 0,C 180,E1 -27941.435,E2 -27941.435} C_VEL
LIN {X 0,Y 72.403,Z 474.611,A -85,B 0,C 180,E1 -27947.204,E2 -27947.204} C_VEL
LIN {X 0,Y 70.582,Z 474.44,A -85,B 0,C 180,E1 -27953.32,E2 -27953.32} C_VEL
LIN {X 0,Y 69.37,Z 473.773,A -85,B 0,C 180,E1 -27959.571,E2 -27959.571} C_VEL
LIN {X 0,Y 68.896,Z 472.539,A -85,B 0,C 180,E1 -27966.592,E2 -27966.592} C_VEL
LIN {X 0,Y 69.469,Z 470.119,A -85,B 0,C 180,E1 -27975.355,E2 -27975.355} C_VEL
LIN {X 0,Y 71.454,Z 466.472,A -85,B 0,C 180,E1 -27984.36,E2 -27984.36} C_VEL
LIN {X 0,Y 74.554,Z 461.65,A -85,B 0,C 180,E1 -27992.706,E2 -27992.706} C_VEL
LIN {X 0,Y 78.859,Z 455.484,A -85,B 0,C 180,E1 -28000.272,E2 -28000.272} C_VEL
LIN {X 0,Y 84.28,Z 447.765,A -85,B 0,C 180,E1 -28006.973,E2 -28006.973} C_VEL
LIN {X 0,Y 89.491,Z 439.867,A -85,B 0,C 180,E1 -28011.906,E2 -28011.906} C_VEL
LIN {X 0,Y 95.304,Z 430.198,A -85,B 0,C 180,E1 -28016.265,E2 -28016.265} C_VEL
LIN {X 0,Y 100.903,Z 419.387,A -85,B 0,C 180,E1 -28019.757,E2 -28019.757} C_VEL
LIN {X 0,Y 106.131,Z 407.328,A -85,B 0,C 180,E1 -28022.554,E2 -28022.554} C_VEL
LIN {X 0,Y 110.135,Z 395.58,A -85,B 0,C 180,E1 -28024.498,E2 -28024.498} C_VEL
LIN {X 0,Y 113.646,Z 382.08,A -85,B 0,C 180,E1 -28026.021,E2 -28026.021} C_VEL
LIN {X 0,Y 115.872,Z 369.157,A -85,B 0,C 180,E1 -28026.943,E2 -28026.943} C_VEL
LIN {X 0,Y 118.647,Z 342.473,A -85,B 0,C 180,E1 -28028.085,E2 -28028.085} C_VEL
LIN {X 0,Y 114.291,Z 332.642,A -85,B 0,C 180,E1 -28032.183,E2 -28032.183} C_VEL
LIN {X 0,Y 110.296,Z 324.863,A -85,B 0,C 180,E1 -28036.504,E2 -28036.504} C_VEL
LIN {X 0,Y 106.821,Z 318.877,A -85,B 0,C 180,E1 -28040.903,E2 -28040.903} C_VEL
LIN {X 0,Y 104.667,Z 315.379,A -85,B 0,C 180,E1 -28044.128,E2 -28044.128} C_VEL
LIN {X 0,Y 102.547,Z 311.929,A -85,B 0,C 180,E1 -28047.951,E2 -28047.951} C_VEL
LIN {X 0,Y 100.375,Z 308.737,A -85,B 0,C 180,E1 -28052.797,E2 -28052.797} C_VEL
LIN {X 0,Y 99.924,Z 307.686,A -85,B 0,C 180,E1 -28054.176,E2 -28054.176} C_VEL
LIN {X 0,Y 97.578,Z 303.996,A -85,B 0,C 180,E1 -28067.536,E2 -28067.536} C_VEL
LIN {X 0,Y 97.764,Z 304.061,A -85,B 0,C 180,E1 -28072.442,E2 -28072.442} C_VEL
LIN {X 0,Y 98.585,Z 305.454,A -85,B 0,C 180,E1 -28077.744,E2 -28077.744} C_VEL
LIN {X 0,Y 100.427,Z 307.925,A -85,B 0,C 180,E1 -28083.901,E2 -28083.901} C_VEL
LIN {X 0,Y 103.181,Z 312.636,A -85,B 0,C 180,E1 -28090.03,E2 -28090.03} C_VEL
LIN {X 0,Y 105.866,Z 317.071,A -85,B 0,C 180,E1 -28094.514,E2 -28094.514} C_VEL
LIN {X 0,Y 109.411,Z 323.001,A -85,B 0,C 180,E1 -28099.224,E2 -28099.224} C_VEL
LIN {X 0,Y 112.748,Z 329.565,A -85,B 0,C 180,E1 -28103.062,E2 -28103.062} C_VEL
LIN {X 0,Y 115.968,Z 336.664,A -85,B 0,C 180,E1 -28106.318,E2 -28106.318} C_VEL
LIN {X 0,Y 118.482,Z 344.786,A -85,B 0,C 180,E1 -28108.884,E2 -28108.884} C_VEL
LIN {X 0,Y 115.374,Z 374.314,A -85,B 0,C 180,E1 -28110.255,E2 -28110.255} C_VEL
LIN {X 0,Y 112.765,Z 387.319,A -85,B 0,C 180,E1 -28111.234,E2 -28111.234} C_VEL
LIN {X 0,Y 109.531,Z 399.024,A -85,B 0,C 180,E1 -28112.627,E2 -28112.627} C_VEL
LIN {X 0,Y 105.494,Z 410.16,A -85,B 0,C 180,E1 -28114.466,E2 -28114.466} C_VEL
LIN {X 0,Y 100.382,Z 421.802,A -85,B 0,C 180,E1 -28117.208,E2 -28117.208} C_VEL
LIN {X 0,Y 95.431,Z 431.187,A -85,B 0,C 180,E1 -28120.172,E2 -28120.172} C_VEL
LIN {X 0,Y 90.348,Z 439.952,A -85,B 0,C 180,E1 -28123.979,E2 -28123.979} C_VEL
LIN {X 0,Y 85.116,Z 447.997,A -85,B 0,C 180,E1 -28128.653,E2 -28128.653} C_VEL
LIN {X 0,Y 79.682,Z 455.853,A -85,B 0,C 180,E1 -28135.014,E2 -28135.014} C_VEL
LIN {X 0,Y 75.193,Z 462.11,A -85,B 0,C 180,E1 -28142.134,E2 -28142.134} C_VEL
LIN {X 0,Y 72.069,Z 467.079,A -85,B 0,C 180,E1 -28150.038,E2 -28150.038} C_VEL
LIN {X 0,Y 70.208,Z 470.885,A -85,B 0,C 180,E1 -28158.446,E2 -28158.446} C_VEL
LIN {X 0,Y 69.603,Z 472.832,A -85,B 0,C 180,E1 -28164.2,E2 -28164.2} C_VEL
LIN {X 0,Y 69.595,Z 474.356,A -85,B 0,C 180,E1 -28169.995,E2 -28169.995} C_VEL
LIN {X 0,Y 69.606,Z 475.409,A -85,B 0,C 180,E1 -28175.79,E2 -28175.79} C_VEL
LIN {X 0,Y 71.411,Z 476.353,A -85,B 0,C 180,E1 -28187.167,E2 -28187.167} C_VEL
LIN {X 0,Y 75.486,Z 475.798,A -85,B 0,C 180,E1 -28197.738,E2 -28197.738} C_VEL
LIN {X 0,Y 81.958,Z 473.661,A -85,B 0,C 180,E1 -28206.883,E2 -28206.883} C_VEL
LIN {X 0,Y 90.167,Z 469.96,A -85,B 0,C 180,E1 -28214.542,E2 -28214.542} C_VEL
LIN {X 0,Y 97.191,Z 466.03,A -85,B 0,C 180,E1 -28219.381,E2 -28219.381} C_VEL
LIN {X 0,Y 104.853,Z 461.005,A -85,B 0,C 180,E1 -28223.539,E2 -28223.539} C_VEL
LIN {X 0,Y 113.035,Z 454.732,A -85,B 0,C 180,E1 -28227.067,E2 -28227.067} C_VEL
LIN {X 0,Y 121.622,Z 446.939,A -85,B 0,C 180,E1 -28230.081,E2 -28230.081} C_VEL
LIN {X 0,Y 129.023,Z 439.044,A -85,B 0,C 180,E1 -28232.263,E2 -28232.263} C_VEL
LIN {X 0,Y 137.41,Z 428.402,A -85,B 0,C 180,E1 -28234.343,E2 -28234.343} C_VEL
LIN {X 0,Y 144.388,Z 417.472,A -85,B 0,C 180,E1 -28235.866,E2 -28235.866} C_VEL
LIN {X 0,Y 150.673,Z 405.192,A -85,B 0,C 180,E1 -28237.098,E2 -28237.098} C_VEL
LIN {X 0,Y 155.417,Z 393.208,A -85,B 0,C 180,E1 -28237.952,E2 -28237.952} C_VEL
LIN {X 0,Y 159.275,Z 379.625,A -85,B 0,C 180,E1 -28238.574,E2 -28238.574} C_VEL
LIN {X 0,Y 160.775,Z 372.033,A -85,B 0,C 180,E1 -28238.899,E2 -28238.899} C_VEL
LIN {X 0,Y 160.029,Z 369.773,A -85,B 0,C 180,E1 -28241.26,E2 -28241.26} C_VEL
LIN {X 0,Y 159.493,Z 367.879,A -85,B 0,C 180,E1 -28243.677,E2 -28243.677} C_VEL
LIN {X 0,Y 159.068,Z 366.23,A -85,B 0,C 180,E1 -28248.484,E2 -28248.484} C_VEL
LIN {X 0,Y 159.129,Z 366.374,A -85,B 0,C 180,E1 -28250.225,E2 -28250.225} C_VEL
LIN {X 0,Y 159.557,Z 367.497,A -85,B 0,C 180,E1 -28253.614,E2 -28253.614} C_VEL
LIN {X 0,Y 159.654,Z 368.608,A -85,B 0,C 180,E1 -28254.514,E2 -28254.514} C_VEL
LIN {X 0,Y 159.481,Z 371.317,A -85,B 0,C 180,E1 -28255.316,E2 -28255.316} C_VEL
LIN {X 0,Y 158.932,Z 375,A -85,B 0,C 180,E1 -28255.829,E2 -28255.829} C_VEL
LIN {X 0,Y 157.621,Z 381.036,A -85,B 0,C 180,E1 -28256.164,E2 -28256.164} C_VEL
LIN {X 0,Y 155.96,Z 387.038,A -85,B 0,C 180,E1 -28256.402,E2 -28256.402} C_VEL
LIN {X 0,Y 151.914,Z 398.565,A -85,B 0,C 180,E1 -28257.067,E2 -28257.067} C_VEL
LIN {X 0,Y 146.791,Z 409.776,A -85,B 0,C 180,E1 -28258.008,E2 -28258.008} C_VEL
LIN {X 0,Y 140.566,Z 420.62,A -85,B 0,C 180,E1 -28259.22,E2 -28259.22} C_VEL
LIN {X 0,Y 133.535,Z 430.614,A -85,B 0,C 180,E1 -28260.7,E2 -28260.7} C_VEL
LIN {X 0,Y 125.552,Z 440.005,A -85,B 0,C 180,E1 -28262.629,E2 -28262.629} C_VEL
LIN {X 0,Y 116.429,Z 448.827,A -85,B 0,C 180,E1 -28265.172,E2 -28265.172} C_VEL
LIN {X 0,Y 106.614,Z 456.75,A -85,B 0,C 180,E1 -28268.607,E2 -28268.607} C_VEL
LIN {X 0,Y 97.944,Z 462.521,A -85,B 0,C 180,E1 -28272.416,E2 -28272.416} C_VEL
LIN {X 0,Y 88.544,Z 467.643,A -85,B 0,C 180,E1 -28277.748,E2 -28277.748} C_VEL
LIN {X 0,Y 83.146,Z 470.098,A -85,B 0,C 180,E1 -28281.61,E2 -28281.61} C_VEL
LIN {X 0,Y 77.264,Z 472.306,A -85,B 0,C 180,E1 -28287.031,E2 -28287.031} C_VEL
LIN {X 0,Y 69.973,Z 474.284,A -85,B 0,C 180,E1 -28296.542,E2 -28296.542} C_VEL
LIN {X 0,Y 66.802,Z 474.676,A -85,B 0,C 180,E1 -28302.578,E2 -28302.578} C_VEL
LIN {X 0,Y 64.152,Z 474.593,A -85,B 0,C 180,E1 -28310.038,E2 -28310.038} C_VEL
LIN {X 0,Y 62.765,Z 474.098,A -85,B 0,C 180,E1 -28315.96,E2 -28315.96} C_VEL
LIN {X 0,Y 61.821,Z 472.664,A -85,B 0,C 180,E1 -28325.373,E2 -28325.373} C_VEL
LIN {X 0,Y 62.592,Z 469.669,A -85,B 0,C 180,E1 -28337.028,E2 -28337.028} C_VEL
LIN {X 0,Y 64.893,Z 465.817,A -85,B 0,C 180,E1 -28346.901,E2 -28346.901} C_VEL
LIN {X 0,Y 68.496,Z 460.777,A -85,B 0,C 180,E1 -28355.894,E2 -28355.894} C_VEL
LIN {X 0,Y 73.4,Z 454.388,A -85,B 0,C 180,E1 -28363.854,E2 -28363.854} C_VEL
LIN {X 0,Y 79.355,Z 446.405,A -85,B 0,C 180,E1 -28370.752,E2 -28370.752} C_VEL
LIN {X 0,Y 85.753,Z 437.098,A -85,B 0,C 180,E1 -28376.237,E2 -28376.237} C_VEL
LIN {X 0,Y 91.967,Z 426.945,A -85,B 0,C 180,E1 -28380.42,E2 -28380.42} C_VEL
LIN {X 0,Y 97.313,Z 416.722,A -85,B 0,C 180,E1 -28383.417,E2 -28383.417} C_VEL
LIN {X 0,Y 102.142,Z 405.577,A -85,B 0,C 180,E1 -28385.796,E2 -28385.796} C_VEL
LIN {X 0,Y 106.452,Z 392.877,A -85,B 0,C 180,E1 -28387.767,E2 -28387.767} C_VEL
LIN {X 0,Y 109.741,Z 379.847,A -85,B 0,C 180,E1 -28389.081,E2 -28389.081} C_VEL
LIN {X 0,Y 111.913,Z 366.645,A -85,B 0,C 180,E1 -28389.893,E2 -28389.893} C_VEL
LIN {X 0,Y 114.153,Z 344.949,A -85,B 0,C 180,E1 -28390.84,E2 -28390.84} C_VEL
LIN {X 0,Y 110.221,Z 335.904,A -85,B 0,C 180,E1 -28395.058,E2 -28395.058} C_VEL
LIN {X 0,Y 106.594,Z 328.528,A -85,B 0,C 180,E1 -28399.602,E2 -28399.602} C_VEL
LIN {X 0,Y 103.144,Z 322.283,A -85,B 0,C 180,E1 -28404.855,E2 -28404.855} C_VEL
LIN {X 0,Y 100.96,Z 318.607,A -85,B 0,C 180,E1 -28409.027,E2 -28409.027} C_VEL
LIN {X 0,Y 98.851,Z 315.144,A -85,B 0,C 180,E1 -28414.321,E2 -28414.321} C_VEL
LIN {X 0,Y 98.498,Z 314.467,A -85,B 0,C 180,E1 -28415.496,E2 -28415.496} C_VEL
LIN {X 0,Y 96.635,Z 311.143,A -85,B 0,C 180,E1 -28427.413,E2 -28427.413} C_VEL
LIN {X 0,Y 96.822,Z 311.142,A -85,B 0,C 180,E1 -28432.409,E2 -28432.409} C_VEL
LIN {X 0,Y 97.612,Z 312.594,A -85,B 0,C 180,E1 -28437.67,E2 -28437.67} C_VEL
LIN {X 0,Y 98.984,Z 314.587,A -85,B 0,C 180,E1 -28442.653,E2 -28442.653} C_VEL
LIN {X 0,Y 101.392,Z 319.049,A -85,B 0,C 180,E1 -28448.617,E2 -28448.617} C_VEL
LIN {X 0,Y 103.873,Z 323.494,A -85,B 0,C 180,E1 -28453.188,E2 -28453.188} C_VEL
LIN {X 0,Y 107.039,Z 329.181,A -85,B 0,C 180,E1 -28457.784,E2 -28457.784} C_VEL
LIN {X 0,Y 110.298,Z 336.095,A -85,B 0,C 180,E1 -28461.862,E2 -28461.862} C_VEL
LIN {X 0,Y 112.482,Z 341.433,A -85,B 0,C 180,E1 -28464.327,E2 -28464.327} C_VEL
LIN {X 0,Y 114.085,Z 346.931,A -85,B 0,C 180,E1 -28466.165,E2 -28466.165} C_VEL
LIN {X 0,Y 111.094,Z 374.033,A -85,B 0,C 180,E1 -28467.396,E2 -28467.396} C_VEL
LIN {X 0,Y 108.522,Z 386.625,A -85,B 0,C 180,E1 -28468.317,E2 -28468.317} C_VEL
LIN {X 0,Y 105.143,Z 398.453,A -85,B 0,C 180,E1 -28469.658,E2 -28469.658} C_VEL
LIN {X 0,Y 100.929,Z 409.717,A -85,B 0,C 180,E1 -28471.454,E2 -28471.454} C_VEL
LIN {X 0,Y 95.564,Z 421.421,A -85,B 0,C 180,E1 -28474.167,E2 -28474.167} C_VEL
LIN {X 0,Y 90.354,Z 430.851,A -85,B 0,C 180,E1 -28477.124,E2 -28477.124} C_VEL
LIN {X 0,Y 84.369,Z 440.555,A -85,B 0,C 180,E1 -28481.43,E2 -28481.43} C_VEL
LIN {X 0,Y 78.854,Z 448.48,A -85,B 0,C 180,E1 -28486.307,E2 -28486.307} C_VEL
LIN {X 0,Y 73.058,Z 456.19,A -85,B 0,C 180,E1 -28493.036,E2 -28493.036} C_VEL
LIN {X 0,Y 67.615,Z 463.276,A -85,B 0,C 180,E1 -28502.107,E2 -28502.107} C_VEL
LIN {X 0,Y 64.533,Z 467.97,A -85,B 0,C 180,E1 -28510.925,E2 -28510.925} C_VEL
LIN {X 0,Y 62.812,Z 471.516,A -85,B 0,C 180,E1 -28520.333,E2 -28520.333} C_VEL
LIN {X 0,Y 62.514,Z 474.03,A -85,B 0,C 180,E1 -28529.995,E2 -28529.995} C_VEL
LIN {X 0,Y 62.553,Z 475.176,A -85,B 0,C 180,E1 -28536.446,E2 -28536.446} C_VEL
LIN {X 0,Y 63.28,Z 475.893,A -85,B 0,C 180,E1 -28542.828,E2 -28542.828} C_VEL
LIN {X 0,Y 66.654,Z 476.193,A -85,B 0,C 180,E1 -28554.94,E2 -28554.94} C_VEL
LIN {X 0,Y 69.255,Z 475.789,A -85,B 0,C 180,E1 -28560.485,E2 -28560.485} C_VEL
LIN {X 0,Y 72.553,Z 475,A -85,B 0,C 180,E1 -28565.529,E2 -28565.529} C_VEL
LIN {X 0,Y 80.643,Z 472.213,A -85,B 0,C 180,E1 -28574.196,E2 -28574.196} C_VEL
LIN {X 0,Y 87.712,Z 469.059,A -85,B 0,C 180,E1 -28579.563,E2 -28579.563} C_VEL
LIN {X 0,Y 95.361,Z 464.905,A -85,B 0,C 180,E1 -28584.157,E2 -28584.157} C_VEL
LIN {X 0,Y 105.049,Z 458.628,A -85,B 0,C 180,E1 -28588.533,E2 -28588.533} C_VEL
LIN {X 0,Y 113.824,Z 451.821,A -85,B 0,C 180,E1 -28591.618,E2 -28591.618} C_VEL
LIN {X 0,Y 121.258,Z 444.953,A -85,B 0,C 180,E1 -28593.937,E2 -28593.937} C_VEL
LIN {X 0,Y 129.037,Z 436.681,A -85,B 0,C 180,E1 -28595.816,E2 -28595.816} C_VEL
LIN {X 0,Y 136.906,Z 426.56,A -85,B 0,C 180,E1 -28597.513,E2 -28597.513} C_VEL
LIN {X 0,Y 144.085,Z 415.244,A -85,B 0,C 180,E1 -28598.877,E2 -28598.877} C_VEL
LIN {X 0,Y 149.716,Z 404.177,A -85,B 0,C 180,E1 -28599.85,E2 -28599.85} C_VEL
LIN {X 0,Y 154.395,Z 392.322,A -85,B 0,C 180,E1 -28600.579,E2 -28600.579} C_VEL
LIN {X 0,Y 158.261,Z 378.711,A -85,B 0,C 180,E1 -28601.13,E2 -28601.13} C_VEL
LIN {X 0,Y 158.634,Z 377.04,A -85,B 0,C 180,E1 -28601.225,E2 -28601.225} C_VEL
LIN {X 0,Y 158.142,Z 374.714,A -85,B 0,C 180,E1 -28604.196,E2 -28604.196} C_VEL
LIN {X 0,Y 157.879,Z 373.276,A -85,B 0,C 180,E1 -28608.318,E2 -28608.318} C_VEL
LIN {X 0,Y 157.924,Z 373.387,A -85,B 0,C 180,E1 -28610.149,E2 -28610.149} C_VEL
LIN {X 0,Y 158.315,Z 374.842,A -85,B 0,C 180,E1 -28613.939,E2 -28613.939} C_VEL
LIN {X 0,Y 158.664,Z 376.593,A -85,B 0,C 180,E1 -28615.996,E2 -28615.996} C_VEL
LIN {X 0,Y 155.96,Z 387.038,A -85,B 0,C 180,E1 -28616.402,E2 -28616.402} C_VEL
LIN {X 0,Y 154.082,Z 392.627,A -85,B 0,C 180,E1 -28616.505,E2 -28616.505} C_VEL
LIN {X 0,Y 150.134,Z 401.633,A -85,B 0,C 180,E1 -28616.024,E2 -28616.024} C_VEL
LIN {X 0,Y 145.518,Z 410.331,A -85,B 0,C 180,E1 -28615.571,E2 -28615.571} C_VEL
LIN {X 0,Y 142.572,Z 415.402,A -85,B 0,C 180,E1 -28615.758,E2 -28615.758} C_VEL
LIN {X 0,Y 135.441,Z 426.286,A -85,B 0,C 180,E1 -28617.016,E2 -28617.016} C_VEL
LIN {X 0,Y 128.302,Z 435.251,A -85,B 0,C 180,E1 -28618.437,E2 -28618.437} C_VEL
LIN {X 0,Y 119.473,Z 444.43,A -85,B 0,C 180,E1 -28620.443,E2 -28620.443} C_VEL
LIN {X 0,Y 109.763,Z 452.735,A -85,B 0,C 180,E1 -28623.09,E2 -28623.09} C_VEL
LIN {X 0,Y 100.721,Z 459.151,A -85,B 0,C 180,E1 -28626.146,E2 -28626.146} C_VEL
LIN {X 0,Y 92.643,Z 463.948,A -85,B 0,C 180,E1 -28629.557,E2 -28629.557} C_VEL
LIN {X 0,Y 83.123,Z 468.608,A -85,B 0,C 180,E1 -28634.676,E2 -28634.676} C_VEL
LIN {X 0,Y 75.059,Z 471.701,A -85,B 0,C 180,E1 -28640.569,E2 -28640.569} C_VEL
LIN {X 0,Y 70.026,Z 473.185,A -85,B 0,C 180,E1 -28645.421,E2 -28645.421} C_VEL
LIN {X 0,Y 63.966,Z 474.465,A -85,B 0,C 180,E1 -28653.296,E2 -28653.296} C_VEL
LIN {X 0,Y 58.66,Z 474.775,A -85,B 0,C 180,E1 -28664.048,E2 -28664.048} C_VEL
LIN {X 0,Y 56.45,Z 474.367,A -85,B 0,C 180,E1 -28671.509,E2 -28671.509} C_VEL
LIN {X 0,Y 54.756,Z 472.779,A -85,B 0,C 180,E1 -28683.895,E2 -28683.895} C_VEL
LIN {X 0,Y 55.76,Z 469.186,A -85,B 0,C 180,E1 -28699.108,E2 -28699.108} C_VEL
LIN {X 0,Y 58.494,Z 465.144,A -85,B 0,C 180,E1 -28710.006,E2 -28710.006} C_VEL
LIN {X 0,Y 62.686,Z 459.901,A -85,B 0,C 180,E1 -28719.687,E2 -28719.687} C_VEL
LIN {X 0,Y 68.209,Z 453.267,A -85,B 0,C 180,E1 -28728.01,E2 -28728.01} C_VEL
LIN {X 0,Y 74.835,Z 444.916,A -85,B 0,C 180,E1 -28735.004,E2 -28735.004} C_VEL
LIN {X 0,Y 81.063,Z 436.332,A -85,B 0,C 180,E1 -28739.928,E2 -28739.928} C_VEL
LIN {X 0,Y 87.073,Z 426.986,A -85,B 0,C 180,E1 -28743.708,E2 -28743.708} C_VEL
LIN {X 0,Y 92.693,Z 416.744,A -85,B 0,C 180,E1 -28746.665,E2 -28746.665} C_VEL
LIN {X 0,Y 97.742,Z 405.584,A -85,B 0,C 180,E1 -28748.992,E2 -28748.992} C_VEL
LIN {X 0,Y 102.26,Z 392.822,A -85,B 0,C 180,E1 -28750.91,E2 -28750.91} C_VEL
LIN {X 0,Y 105.604,Z 380.081,A -85,B 0,C 180,E1 -28752.146,E2 -28752.146} C_VEL
LIN {X 0,Y 107.978,Z 366.142,A -85,B 0,C 180,E1 -28752.95,E2 -28752.95} C_VEL
LIN {X 0,Y 109.939,Z 347.729,A -85,B 0,C 180,E1 -28753.739,E2 -28753.739} C_VEL
LIN {X 0,Y 106.498,Z 339.392,A -85,B 0,C 180,E1 -28758.042,E2 -28758.042} C_VEL
LIN {X 0,Y 103.555,Z 333.25,A -85,B 0,C 180,E1 -28762.262,E2 -28762.262} C_VEL
LIN {X 0,Y 100.839,Z 328.004,A -85,B 0,C 180,E1 -28767.081,E2 -28767.081} C_VEL
LIN {X 0,Y 99.168,Z 324.959,A -85,B 0,C 180,E1 -28770.682,E2 -28770.682} C_VEL
LIN {X 0,Y 97.238,Z 321.305,A -85,B 0,C 180,E1 -28776.475,E2 -28776.475} C_VEL
LIN {X 0,Y 95.689,Z 318.305,A -85,B 0,C 180,E1 -28787.286,E2 -28787.286} C_VEL
LIN {X 0,Y 95.876,Z 318.215,A -85,B 0,C 180,E1 -28792.333,E2 -28792.333} C_VEL
LIN {X 0,Y 96.496,Z 319.503,A -85,B 0,C 180,E1 -28796.921,E2 -28796.921} C_VEL
LIN {X 0,Y 97.642,Z 321.376,A -85,B 0,C 180,E1 -28801.562,E2 -28801.562} C_VEL
LIN {X 0,Y 99.684,Z 325.545,A -85,B 0,C 180,E1 -28807.252,E2 -28807.252} C_VEL
LIN {X 0,Y 102.016,Z 330.021,A -85,B 0,C 180,E1 -28811.941,E2 -28811.941} C_VEL
LIN {X 0,Y 105.308,Z 336.61,A -85,B 0,C 180,E1 -28817.13,E2 -28817.13} C_VEL
LIN {X 0,Y 108.744,Z 344.834,A -85,B 0,C 180,E1 -28821.682,E2 -28821.682} C_VEL
LIN {X 0,Y 109.872,Z 349.006,A -85,B 0,C 180,E1 -28823.197,E2 -28823.197} C_VEL
LIN {X 0,Y 107.023,Z 374.031,A -85,B 0,C 180,E1 -28824.347,E2 -28824.347} C_VEL
LIN {X 0,Y 104.212,Z 387.094,A -85,B 0,C 180,E1 -28825.254,E2 -28825.254} C_VEL
LIN {X 0,Y 100.681,Z 398.866,A -85,B 0,C 180,E1 -28826.566,E2 -28826.566} C_VEL
LIN {X 0,Y 95.961,Z 410.793,A -85,B 0,C 180,E1 -28828.489,E2 -28828.489} C_VEL
LIN {X 0,Y 90.327,Z 422.267,A -85,B 0,C 180,E1 -28831.138,E2 -28831.138} C_VEL
LIN {X 0,Y 84.252,Z 432.622,A -85,B 0,C 180,E1 -28834.533,E2 -28834.533} C_VEL
LIN {X 0,Y 78.325,Z 441.451,A -85,B 0,C 180,E1 -28838.697,E2 -28838.697} C_VEL
LIN {X 0,Y 72.739,Z 448.9,A -85,B 0,C 180,E1 -28843.555,E2 -28843.555} C_VEL
LIN {X 0,Y 66.535,Z 456.509,A -85,B 0,C 180,E1 -28850.665,E2 -28850.665} C_VEL
LIN {X 0,Y 61.399,Z 462.6,A -85,B 0,C 180,E1 -28858.991,E2 -28858.991} C_VEL
LIN {X 0,Y 57.855,Z 467.419,A -85,B 0,C 180,E1 -28868.622,E2 -28868.622} C_VEL
LIN {X 0,Y 55.836,Z 471.081,A -85,B 0,C 180,E1 -28879.111,E2 -28879.111} C_VEL
LIN {X 0,Y 55.415,Z 473.701,A -85,B 0,C 180,E1 -28889.994,E2 -28889.994} C_VEL
LIN {X 0,Y 55.521,Z 474.905,A -85,B 0,C 180,E1 -28897.266,E2 -28897.266} C_VEL
LIN {X 0,Y 56.364,Z 475.713,A -85,B 0,C 180,E1 -28904.434,E2 -28904.434} C_VEL
LIN {X 0,Y 60.264,Z 476.121,A -85,B 0,C 180,E1 -28917.8,E2 -28917.8} C_VEL
LIN {X 0,Y 66.906,Z 475.055,A -85,B 0,C 180,E1 -28929.062,E2 -28929.062} C_VEL
LIN {X 0,Y 71.112,Z 473.947,A -85,B 0,C 180,E1 -28933.766,E2 -28933.766} C_VEL
LIN {X 0,Y 80.676,Z 470.493,A -85,B 0,C 180,E1 -28941.623,E2 -28941.623} C_VEL
LIN {X 0,Y 87.684,Z 467.285,A -85,B 0,C 180,E1 -28945.853,E2 -28945.853} C_VEL
LIN {X 0,Y 97.129,Z 462.049,A -85,B 0,C 180,E1 -28950.253,E2 -28950.253} C_VEL
LIN {X 0,Y 106.042,Z 456.103,A -85,B 0,C 180,E1 -28953.465,E2 -28953.465} C_VEL
LIN {X 0,Y 115.249,Z 448.752,A -85,B 0,C 180,E1 -28956.157,E2 -28956.157} C_VEL
LIN {X 0,Y 123.122,Z 441.284,A -85,B 0,C 180,E1 -28958.052,E2 -28958.052} C_VEL
LIN {X 0,Y 131.159,Z 432.27,A -85,B 0,C 180,E1 -28959.663,E2 -28959.663} C_VEL
LIN {X 0,Y 138.461,Z 422.329,A -85,B 0,C 180,E1 -28960.965,E2 -28960.965} C_VEL
LIN {X 0,Y 145.001,Z 411.405,A -85,B 0,C 180,E1 -28962.017,E2 -28962.017} C_VEL
LIN {X 0,Y 150.72,Z 399.364,A -85,B 0,C 180,E1 -28962.869,E2 -28962.869} C_VEL
LIN {X 0,Y 155.24,Z 386.74,A -85,B 0,C 180,E1 -28963.408,E2 -28963.408} C_VEL
LIN {X 0,Y 156.517,Z 382.224,A -85,B 0,C 180,E1 -28963.607,E2 -28963.607} C_VEL
LIN {X 0,Y 156.385,Z 381.224,A -85,B 0,C 180,E1 -28965.349,E2 -28965.349} C_VEL
LIN {X 0,Y 156.295,Z 380.326,A -85,B 0,C 180,E1 -28968.197,E2 -28968.197} C_VEL
LIN {X 0,Y 156.338,Z 380.351,A -85,B 0,C 180,E1 -28970.048,E2 -28970.048} C_VEL
LIN {X 0,Y 156.569,Z 381.61,A -85,B 0,C 180,E1 -28973.408,E2 -28973.408} C_VEL
LIN {X 0,Y 156.577,Z 381.741,A -85,B 0,C 180,E1 -28973.581,E2 -28973.581} C_VEL
LIN {X 0,Y 152.553,Z 394.425,A -85,B 0,C 180,E1 -28974.171,E2 -28974.171} C_VEL
LIN {X 0,Y 147.267,Z 406.691,A -85,B 0,C 180,E1 -28974.98,E2 -28974.98} C_VEL
LIN {X 0,Y 142.572,Z 415.402,A -85,B 0,C 180,E1 -28975.758,E2 -28975.758} C_VEL
LIN {X 0,Y 140.426,Z 418.796,A -85,B 0,C 180,E1 -28975.825,E2 -28975.825} C_VEL
LIN {X 0,Y 132.361,Z 429.257,A -85,B 0,C 180,E1 -28974.667,E2 -28974.667} C_VEL
LIN {X 0,Y 129.803,Z 432.293,A -85,B 0,C 180,E1 -28974.788,E2 -28974.788} C_VEL
LIN {X 0,Y 121.291,Z 441.459,A -85,B 0,C 180,E1 -28976.377,E2 -28976.377} C_VEL
LIN {X 0,Y 112.492,Z 449.344,A -85,B 0,C 180,E1 -28978.277,E2 -28978.277} C_VEL
LIN {X 0,Y 103.662,Z 455.967,A -85,B 0,C 180,E1 -28980.589,E2 -28980.589} C_VEL
LIN {X 0,Y 95.113,Z 461.341,A -85,B 0,C 180,E1 -28983.349,E2 -28983.349} C_VEL
LIN {X 0,Y 85.052,Z 466.536,A -85,B 0,C 180,E1 -28987.474,E2 -28987.474} C_VEL
LIN {X 0,Y 75.617,Z 470.372,A -85,B 0,C 180,E1 -28992.628,E2 -28992.628} C_VEL
LIN {X 0,Y 66.978,Z 472.998,A -85,B 0,C 180,E1 -28999.217,E2 -28999.217} C_VEL
LIN {X 0,Y 58.765,Z 474.58,A -85,B 0,C 180,E1 -29008.552,E2 -29008.552} C_VEL
LIN {X 0,Y 53.466,Z 474.926,A -85,B 0,C 180,E1 -29017.948,E2 -29017.948} C_VEL
LIN {X 0,Y 50.534,Z 474.6,A -85,B 0,C 180,E1 -29025.953,E2 -29025.953} C_VEL
LIN {X 0,Y 47.769,Z 472.889,A -85,B 0,C 180,E1 -29041.912,E2 -29041.912} C_VEL
LIN {X 0,Y 48.285,Z 469.833,A -85,B 0,C 180,E1 -29057.396,E2 -29057.396} C_VEL
LIN {X 0,Y 51.018,Z 465.964,A -85,B 0,C 180,E1 -29070.007,E2 -29070.007} C_VEL
LIN {X 0,Y 55.417,Z 460.908,A -85,B 0,C 180,E1 -29080.972,E2 -29080.972} C_VEL
LIN {X 0,Y 61.249,Z 454.513,A -85,B 0,C 180,E1 -29090.141,E2 -29090.141} C_VEL
LIN {X 0,Y 68.243,Z 446.506,A -85,B 0,C 180,E1 -29097.614,E2 -29097.614} C_VEL
LIN {X 0,Y 75.698,Z 436.974,A -85,B 0,C 180,E1 -29103.359,E2 -29103.359} C_VEL
LIN {X 0,Y 82.498,Z 427.016,A -85,B 0,C 180,E1 -29107.376,E2 -29107.376} C_VEL
LIN {X 0,Y 88.409,Z 416.755,A -85,B 0,C 180,E1 -29110.237,E2 -29110.237} C_VEL
LIN {X 0,Y 93.688,Z 405.58,A -85,B 0,C 180,E1 -29112.469,E2 -29112.469} C_VEL
LIN {X 0,Y 98.375,Z 392.857,A -85,B 0,C 180,E1 -29114.295,E2 -29114.295} C_VEL
LIN {X 0,Y 101.944,Z 379.608,A -85,B 0,C 180,E1 -29115.499,E2 -29115.499} C_VEL
LIN {X 0,Y 104.263,Z 366.296,A -85,B 0,C 180,E1 -29116.22,E2 -29116.22} C_VEL
LIN {X 0,Y 106.002,Z 350.542,A -85,B 0,C 180,E1 -29116.884,E2 -29116.884} C_VEL
LIN {X 0,Y 102.983,Z 342.964,A -85,B 0,C 180,E1 -29121.248,E2 -29121.248} C_VEL
LIN {X 0,Y 100.559,Z 337.505,A -85,B 0,C 180,E1 -29125.453,E2 -29125.453} C_VEL
LIN {X 0,Y 98.389,Z 333.106,A -85,B 0,C 180,E1 -29130.016,E2 -29130.016} C_VEL
LIN {X 0,Y 97.525,Z 331.415,A -85,B 0,C 180,E1 -29132.225,E2 -29132.225} C_VEL
LIN {X 0,Y 95.93,Z 328.081,A -85,B 0,C 180,E1 -29137.739,E2 -29137.739} C_VEL
LIN {X 0,Y 94.757,Z 325.268,A -85,B 0,C 180,E1 -29148.198,E2 -29148.198} C_VEL
LIN {X 0,Y 94.928,Z 325.29,A -85,B 0,C 180,E1 -29152.256,E2 -29152.256} C_VEL
LIN {X 0,Y 95.455,Z 326.576,A -85,B 0,C 180,E1 -29156.523,E2 -29156.523} C_VEL
LIN {X 0,Y 96.355,Z 328.204,A -85,B 0,C 180,E1 -29160.513,E2 -29160.513} C_VEL
LIN {X 0,Y 97.974,Z 331.898,A -85,B 0,C 180,E1 -29165.677,E2 -29165.677} C_VEL
LIN {X 0,Y 100.001,Z 336.134,A -85,B 0,C 180,E1 -29170.237,E2 -29170.237} C_VEL
LIN {X 0,Y 102.74,Z 342.165,A -85,B 0,C 180,E1 -29175.149,E2 -29175.149} C_VEL
LIN {X 0,Y 105.696,Z 349.995,A -85,B 0,C 180,E1 -29179.568,E2 -29179.568} C_VEL
LIN {X 0,Y 105.992,Z 351.14,A -85,B 0,C 180,E1 -29180.027,E2 -29180.027} C_VEL
LIN {X 0,Y 103.235,Z 374.302,A -85,B 0,C 180,E1 -29181.088,E2 -29181.088} C_VEL
LIN {X 0,Y 100.461,Z 386.723,A -85,B 0,C 180,E1 -29181.886,E2 -29181.886} C_VEL
LIN {X 0,Y 96.942,Z 398.189,A -85,B 0,C 180,E1 -29183.095,E2 -29183.095} C_VEL
LIN {X 0,Y 92.009,Z 410.27,A -85,B 0,C 180,E1 -29184.89,E2 -29184.89} C_VEL
LIN {X 0,Y 86.118,Z 421.824,A -85,B 0,C 180,E1 -29187.433,E2 -29187.433} C_VEL
LIN {X 0,Y 79.716,Z 432.244,A -85,B 0,C 180,E1 -29190.722,E2 -29190.722} C_VEL
LIN {X 0,Y 72.767,Z 441.938,A -85,B 0,C 180,E1 -29195.294,E2 -29195.294} C_VEL
LIN {X 0,Y 66.823,Z 449.305,A -85,B 0,C 180,E1 -29200.307,E2 -29200.307} C_VEL
LIN {X 0,Y 60.137,Z 456.818,A -85,B 0,C 180,E1 -29207.773,E2 -29207.773} C_VEL
LIN {X 0,Y 53.827,Z 463.719,A -85,B 0,C 180,E1 -29218.509,E2 -29218.509} C_VEL
LIN {X 0,Y 50.289,Z 468.259,A -85,B 0,C 180,E1 -29229.544,E2 -29229.544} C_VEL
LIN {X 0,Y 48.454,Z 471.675,A -85,B 0,C 180,E1 -29241.653,E2 -29241.653} C_VEL
LIN {X 0,Y 48.332,Z 473.362,A -85,B 0,C 180,E1 -29249.993,E2 -29249.993} C_VEL
LIN {X 0,Y 48.49,Z 474.617,A -85,B 0,C 180,E1 -29258.327,E2 -29258.327} C_VEL
LIN {X 0,Y 51.398,Z 475.973,A -85,B 0,C 180,E1 -29274.211,E2 -29274.211} C_VEL
LIN {X 0,Y 57.429,Z 475.754,A -85,B 0,C 180,E1 -29287.718,E2 -29287.718} C_VEL
LIN {X 0,Y 66.157,Z 474.06,A -85,B 0,C 180,E1 -29298.033,E2 -29298.033} C_VEL
LIN {X 0,Y 71.134,Z 472.63,A -85,B 0,C 180,E1 -29302.214,E2 -29302.214} C_VEL
LIN {X 0,Y 82.057,Z 468.504,A -85,B 0,C 180,E1 -29308.914,E2 -29308.914} C_VEL
LIN {X 0,Y 90.787,Z 464.261,A -85,B 0,C 180,E1 -29312.894,E2 -29312.894} C_VEL
LIN {X 0,Y 101.507,Z 457.895,A -85,B 0,C 180,E1 -29316.537,E2 -29316.537} C_VEL
LIN {X 0,Y 111.023,Z 450.95,A -85,B 0,C 180,E1 -29319.01,E2 -29319.01} C_VEL
LIN {X 0,Y 115.77,Z 446.905,A -85,B 0,C 180,E1 -29320.203,E2 -29320.203} C_VEL
LIN {X 0,Y 125.592,Z 437.328,A -85,B 0,C 180,E1 -29322.036,E2 -29322.036} C_VEL
LIN {X 0,Y 133.852,Z 427.487,A -85,B 0,C 180,E1 -29323.371,E2 -29323.371} C_VEL
LIN {X 0,Y 141.338,Z 416.445,A -85,B 0,C 180,E1 -29324.444,E2 -29324.444} C_VEL
LIN {X 0,Y 147.566,Z 404.971,A -85,B 0,C 180,E1 -29325.252,E2 -29325.252} C_VEL
LIN {X 0,Y 152.237,Z 393.984,A -85,B 0,C 180,E1 -29325.792,E2 -29325.792} C_VEL
LIN {X 0,Y 154.227,Z 388.258,A -85,B 0,C 180,E1 -29325.978,E2 -29325.978} C_VEL
LIN {X 0,Y 154.335,Z 387.597,A -85,B 0,C 180,E1 -29326.83,E2 -29326.83} C_VEL
LIN {X 0,Y 154.417,Z 387.016,A -85,B 0,C 180,E1 -29329.502,E2 -29329.502} C_VEL
LIN {X 0,Y 154.066,Z 388.579,A -85,B 0,C 180,E1 -29331.239,E2 -29331.239} C_VEL
LIN {X 0,Y 149.08,Z 401.53,A -85,B 0,C 180,E1 -29331.868,E2 -29331.868} C_VEL
LIN {X 0,Y 143.489,Z 412.624,A -85,B 0,C 180,E1 -29332.649,E2 -29332.649} C_VEL
LIN {X 0,Y 136.913,Z 423.056,A -85,B 0,C 180,E1 -29333.637,E2 -29333.637} C_VEL
LIN {X 0,Y 129.803,Z 432.293,A -85,B 0,C 180,E1 -29334.788,E2 -29334.788} C_VEL
LIN {X 0,Y 125.864,Z 436.676,A -85,B 0,C 180,E1 -29335.16,E2 -29335.16} C_VEL
LIN {X 0,Y 118.674,Z 443.575,A -85,B 0,C 180,E1 -29335.067,E2 -29335.067} C_VEL
LIN {X 0,Y 111.04,Z 449.822,A -85,B 0,C 180,E1 -29335.064,E2 -29335.064} C_VEL
LIN {X 0,Y 106.43,Z 453.226,A -85,B 0,C 180,E1 -29335.668,E2 -29335.668} C_VEL
LIN {X 0,Y 96.682,Z 459.585,A -85,B 0,C 180,E1 -29338.091,E2 -29338.091} C_VEL
LIN {X 0,Y 87.399,Z 464.55,A -85,B 0,C 180,E1 -29341.01,E2 -29341.01} C_VEL
LIN {X 0,Y 77.232,Z 468.924,A -85,B 0,C 180,E1 -29345.203,E2 -29345.203} C_VEL
LIN {X 0,Y 71.038,Z 471.019,A -85,B 0,C 180,E1 -29348.416,E2 -29348.416} C_VEL
LIN {X 0,Y 64.792,Z 472.759,A -85,B 0,C 180,E1 -29352.543,E2 -29352.543} C_VEL
LIN {X 0,Y 58.954,Z 474.011,A -85,B 0,C 180,E1 -29357.526,E2 -29357.526} C_VEL
LIN {X 0,Y 53.638,Z 474.741,A -85,B 0,C 180,E1 -29363.498,E2 -29363.498} C_VEL
LIN {X 0,Y 48.991,Z 475.028,A -85,B 0,C 180,E1 -29370.615,E2 -29370.615} C_VEL
LIN {X 0,Y 45.226,Z 474.832,A -85,B 0,C 180,E1 -29379.027,E2 -29379.027} C_VEL
LIN {X 0,Y 42.433,Z 474.153,A -85,B 0,C 180,E1 -29388.52,E2 -29388.52} C_VEL
LIN {X 0,Y 40.839,Z 472.994,A -85,B 0,C 180,E1 -29399.297,E2 -29399.297} C_VEL
LIN {X 0,Y 40.85,Z 470.451,A -85,B 0,C 180,E1 -29415.053,E2 -29415.053} C_VEL
LIN {X 0,Y 43.509,Z 466.763,A -85,B 0,C 180,E1 -29430.008,E2 -29430.008} C_VEL
LIN {X 0,Y 48.154,Z 461.892,A -85,B 0,C 180,E1 -29442.653,E2 -29442.653} C_VEL
LIN {X 0,Y 54.393,Z 455.693,A -85,B 0,C 180,E1 -29452.813,E2 -29452.813} C_VEL
LIN {X 0,Y 61.824,Z 447.947,A -85,B 0,C 180,E1 -29460.773,E2 -29460.773} C_VEL
LIN {X 0,Y 68.7,Z 440.011,A -85,B 0,C 180,E1 -29466.037,E2 -29466.037} C_VEL
LIN {X 0,Y 76.025,Z 430.283,A -85,B 0,C 180,E1 -29470.329,E2 -29470.329} C_VEL
LIN {X 0,Y 82.925,Z 419.406,A -85,B 0,C 180,E1 -29473.525,E2 -29473.525} C_VEL
LIN {X 0,Y 88.439,Z 408.901,A -85,B 0,C 180,E1 -29475.665,E2 -29475.665} C_VEL
LIN {X 0,Y 93.271,Z 397.307,A -85,B 0,C 180,E1 -29477.395,E2 -29477.395} C_VEL
LIN {X 0,Y 97.323,Z 384.321,A -85,B 0,C 180,E1 -29478.688,E2 -29478.688} C_VEL
LIN {X 0,Y 100.177,Z 370.928,A -85,B 0,C 180,E1 -29479.541,E2 -29479.541} C_VEL
LIN {X 0,Y 102.331,Z 353.464,A -85,B 0,C 180,E1 -29480.22,E2 -29480.22} C_VEL
LIN {X 0,Y 99.734,Z 346.484,A -85,B 0,C 180,E1 -29484.794,E2 -29484.794} C_VEL
LIN {X 0,Y 97.456,Z 341.049,A -85,B 0,C 180,E1 -29489.699,E2 -29489.699} C_VEL
LIN {X 0,Y 96.021,Z 337.956,A -85,B 0,C 180,E1 -29493.63,E2 -29493.63} C_VEL
LIN {X 0,Y 94.735,Z 334.927,A -85,B 0,C 180,E1 -29498.687,E2 -29498.687} C_VEL
LIN {X 0,Y 93.832,Z 332.23,A -85,B 0,C 180,E1 -29509.126,E2 -29509.126} C_VEL
LIN {X 0,Y 93.98,Z 332.365,A -85,B 0,C 180,E1 -29512.178,E2 -29512.178} C_VEL
LIN {X 0,Y 95.023,Z 334.724,A -85,B 0,C 180,E1 -29519.032,E2 -29519.032} C_VEL
LIN {X 0,Y 96.441,Z 338.502,A -85,B 0,C 180,E1 -29524.354,E2 -29524.354} C_VEL
LIN {X 0,Y 98.239,Z 342.672,A -85,B 0,C 180,E1 -29528.888,E2 -29528.888} C_VEL
LIN {X 0,Y 100.478,Z 348.228,A -85,B 0,C 180,E1 -29533.408,E2 -29533.408} C_VEL
LIN {X 0,Y 102.374,Z 353.747,A -85,B 0,C 180,E1 -29536.7,E2 -29536.7} C_VEL
LIN {X 0,Y 99.839,Z 374.015,A -85,B 0,C 180,E1 -29537.575,E2 -29537.575} C_VEL
LIN {X 0,Y 96.831,Z 387.055,A -85,B 0,C 180,E1 -29538.343,E2 -29538.343} C_VEL
LIN {X 0,Y 93.174,Z 398.42,A -85,B 0,C 180,E1 -29539.452,E2 -29539.452} C_VEL
LIN {X 0,Y 88.452,Z 409.609,A -85,B 0,C 180,E1 -29540.988,E2 -29540.988} C_VEL
LIN {X 0,Y 83.085,Z 419.976,A -85,B 0,C 180,E1 -29543.08,E2 -29543.08} C_VEL
LIN {X 0,Y 77.805,Z 428.531,A -85,B 0,C 180,E1 -29545.399,E2 -29545.399} C_VEL
LIN {X 0,Y 70.42,Z 438.735,A -85,B 0,C 180,E1 -29549.444,E2 -29549.444} C_VEL
LIN {X 0,Y 63.459,Z 447.009,A -85,B 0,C 180,E1 -29554.308,E2 -29554.308} C_VEL
LIN {X 0,Y 56.19,Z 454.8,A -85,B 0,C 180,E1 -29561.362,E2 -29561.362} C_VEL
LIN {X 0,Y 49.738,Z 461.196,A -85,B 0,C 180,E1 -29570.509,E2 -29570.509} C_VEL
LIN {X 0,Y 44.864,Z 466.266,A -85,B 0,C 180,E1 -29581.96,E2 -29581.96} C_VEL
LIN {X 0,Y 41.975,Z 470.171,A -85,B 0,C 180,E1 -29595.446,E2 -29595.446} C_VEL
LIN {X 0,Y 41.226,Z 473.015,A -85,B 0,C 180,E1 -29609.992,E2 -29609.992} C_VEL
LIN {X 0,Y 41.472,Z 474.326,A -85,B 0,C 180,E1 -29619.748,E2 -29619.748} C_VEL
LIN {X 0,Y 42.76,Z 475.251,A -85,B 0,C 180,E1 -29629.183,E2 -29629.183} C_VEL
LIN {X 0,Y 48.11,Z 475.972,A -85,B 0,C 180,E1 -29645.747,E2 -29645.747} C_VEL
LIN {X 0,Y 56.567,Z 475.138,A -85,B 0,C 180,E1 -29658.189,E2 -29658.189} C_VEL
LIN {X 0,Y 67.015,Z 472.822,A -85,B 0,C 180,E1 -29667.022,E2 -29667.022} C_VEL
LIN {X 0,Y 75.667,Z 470.009,A -85,B 0,C 180,E1 -29671.919,E2 -29671.919} C_VEL
LIN {X 0,Y 84.683,Z 466.238,A -85,B 0,C 180,E1 -29675.899,E2 -29675.899} C_VEL
LIN {X 0,Y 94.123,Z 461.392,A -85,B 0,C 180,E1 -29678.952,E2 -29678.952} C_VEL
LIN {X 0,Y 103.796,Z 455.355,A -85,B 0,C 180,E1 -29681.419,E2 -29681.419} C_VEL
LIN {X 0,Y 113.581,Z 447.928,A -85,B 0,C 180,E1 -29683.542,E2 -29683.542} C_VEL
LIN {X 0,Y 123.615,Z 438.599,A -85,B 0,C 180,E1 -29685.119,E2 -29685.119} C_VEL
LIN {X 0,Y 132.865,Z 428.006,A -85,B 0,C 180,E1 -29686.386,E2 -29686.386} C_VEL
LIN {X 0,Y 140.478,Z 417.135,A -85,B 0,C 180,E1 -29687.295,E2 -29687.295} C_VEL
LIN {X 0,Y 146.944,Z 405.556,A -85,B 0,C 180,E1 -29687.986,E2 -29687.986} C_VEL
LIN {X 0,Y 150.684,Z 397.281,A -85,B 0,C 180,E1 -29688.351,E2 -29688.351} C_VEL
LIN {X 0,Y 150.368,Z 398.053,A -85,B 0,C 180,E1 -29688.952,E2 -29688.952} C_VEL
LIN {X 0,Y 144.414,Z 410.369,A -85,B 0,C 180,E1 -29689.632,E2 -29689.632} C_VEL
LIN {X 0,Y 137.148,Z 422.098,A -85,B 0,C 180,E1 -29690.537,E2 -29690.537} C_VEL
LIN {X 0,Y 129.488,Z 432.039,A -85,B 0,C 180,E1 -29691.579,E2 -29691.579} C_VEL
LIN {X 0,Y 120.366,Z 441.661,A -85,B 0,C 180,E1 -29693.001,E2 -29693.001} C_VEL
LIN {X 0,Y 111.163,Z 449.659,A -85,B 0,C 180,E1 -29694.679,E2 -29694.679} C_VEL
LIN {X 0,Y 106.43,Z 453.226,A -85,B 0,C 180,E1 -29695.668,E2 -29695.668} C_VEL
LIN {X 0,Y 101.65,Z 456.469,A -85,B 0,C 180,E1 -29696.376,E2 -29696.376} C_VEL
LIN {X 0,Y 93.037,Z 461.366,A -85,B 0,C 180,E1 -29696.755,E2 -29696.755} C_VEL
LIN {X 0,Y 84.121,Z 465.567,A -85,B 0,C 180,E1 -29697.343,E2 -29697.343} C_VEL
LIN {X 0,Y 78.909,Z 467.672,A -85,B 0,C 180,E1 -29698.569,E2 -29698.569} C_VEL
LIN {X 0,Y 70.316,Z 470.686,A -85,B 0,C 180,E1 -29701.99,E2 -29701.99} C_VEL
LIN {X 0,Y 61.925,Z 472.891,A -85,B 0,C 180,E1 -29706.494,E2 -29706.494} C_VEL
LIN {X 0,Y 50.987,Z 474.732,A -85,B 0,C 180,E1 -29715.256,E2 -29715.256} C_VEL
LIN {X 0,Y 45.457,Z 475.098,A -85,B 0,C 180,E1 -29721.952,E2 -29721.952} C_VEL
LIN {X 0,Y 40.067,Z 474.977,A -85,B 0,C 180,E1 -29731.709,E2 -29731.709} C_VEL
LIN {X 0,Y 36.921,Z 474.459,A -85,B 0,C 180,E1 -29740.426,E2 -29740.426} C_VEL
LIN {X 0,Y 34.009,Z 473.084,A -85,B 0,C 180,E1 -29755.676,E2 -29755.676} C_VEL
LIN {X 0,Y 33.989,Z 469.955,A -85,B 0,C 180,E1 -29778.077,E2 -29778.077} C_VEL
LIN {X 0,Y 37.39,Z 466.059,A -85,B 0,C 180,E1 -29795.402,E2 -29795.402} C_VEL
LIN {X 0,Y 43,Z 460.972,A -85,B 0,C 180,E1 -29809.088,E2 -29809.088} C_VEL
LIN {X 0,Y 50.188,Z 454.543,A -85,B 0,C 180,E1 -29819.356,E2 -29819.356} C_VEL
LIN {X 0,Y 57.04,Z 447.943,A -85,B 0,C 180,E1 -29825.828,E2 -29825.828} C_VEL
LIN {X 0,Y 64.418,Z 439.982,A -85,B 0,C 180,E1 -29830.896,E2 -29830.896} C_VEL
LIN {X 0,Y 72.169,Z 430.213,A -85,B 0,C 180,E1 -29834.918,E2 -29834.918} C_VEL
LIN {X 0,Y 79.375,Z 419.31,A -85,B 0,C 180,E1 -29837.868,E2 -29837.868} C_VEL
LIN {X 0,Y 85.271,Z 408.441,A -85,B 0,C 180,E1 -29839.863,E2 -29839.863} C_VEL
LIN {X 0,Y 90.446,Z 396.142,A -85,B 0,C 180,E1 -29841.488,E2 -29841.488} C_VEL
LIN {X 0,Y 94.683,Z 382.625,A -85,B 0,C 180,E1 -29842.626,E2 -29842.626} C_VEL
LIN {X 0,Y 97.356,Z 369.71,A -85,B 0,C 180,E1 -29843.306,E2 -29843.306} C_VEL
LIN {X 0,Y 98.992,Z 357.146,A -85,B 0,C 180,E1 -29843.694,E2 -29843.694} C_VEL
LIN {X 0,Y 98.843,Z 356.122,A -85,B 0,C 180,E1 -29844.103,E2 -29844.103} C_VEL
LIN {X 0,Y 97.066,Z 350.933,A -85,B 0,C 180,E1 -29847.953,E2 -29847.953} C_VEL
LIN {X 0,Y 95.325,Z 346.393,A -85,B 0,C 180,E1 -29852.547,E2 -29852.547} C_VEL
LIN {X 0,Y 94.455,Z 344.218,A -85,B 0,C 180,E1 -29855.53,E2 -29855.53} C_VEL
LIN {X 0,Y 93.551,Z 341.741,A -85,B 0,C 180,E1 -29859.744,E2 -29859.744} C_VEL
LIN {X 0,Y 92.908,Z 339.247,A -85,B 0,C 180,E1 -29869.556,E2 -29869.556} C_VEL
LIN {X 0,Y 93.092,Z 339.603,A -85,B 0,C 180,E1 -29872.873,E2 -29872.873} C_VEL
LIN {X 0,Y 93.811,Z 341.611,A -85,B 0,C 180,E1 -29878.029,E2 -29878.029} C_VEL
LIN {X 0,Y 94.928,Z 345.006,A -85,B 0,C 180,E1 -29882.873,E2 -29882.873} C_VEL
LIN {X 0,Y 96.595,Z 349.39,A -85,B 0,C 180,E1 -29887.672,E2 -29887.672} C_VEL
LIN {X 0,Y 98.451,Z 354.763,A -85,B 0,C 180,E1 -29891.89,E2 -29891.89} C_VEL
LIN {X 0,Y 99.019,Z 356.689,A -85,B 0,C 180,E1 -29893.084,E2 -29893.084} C_VEL
LIN {X 0,Y 96.846,Z 373.633,A -85,B 0,C 180,E1 -29893.829,E2 -29893.829} C_VEL
LIN {X 0,Y 93.703,Z 386.976,A -85,B 0,C 180,E1 -29894.521,E2 -29894.521} C_VEL
LIN {X 0,Y 89.819,Z 398.624,A -85,B 0,C 180,E1 -29895.537,E2 -29895.537} C_VEL
LIN {X 0,Y 84.546,Z 410.532,A -85,B 0,C 180,E1 -29897.058,E2 -29897.058} C_VEL
LIN {X 0,Y 78.138,Z 421.98,A -85,B 0,C 180,E1 -29899.184,E2 -29899.184} C_VEL
LIN {X 0,Y 71.127,Z 432.341,A -85,B 0,C 180,E1 -29902.119,E2 -29902.119} C_VEL
LIN {X 0,Y 62.884,Z 442.46,A -85,B 0,C 180,E1 -29906.598,E2 -29906.598} C_VEL
LIN {X 0,Y 54.397,Z 451.338,A -85,B 0,C 180,E1 -29912.871,E2 -29912.871} C_VEL
LIN {X 0,Y 46.799,Z 458.416,A -85,B 0,C 180,E1 -29921.324,E2 -29921.324} C_VEL
LIN {X 0,Y 40.42,Z 464.045,A -85,B 0,C 180,E1 -29932.504,E2 -29932.504} C_VEL
LIN {X 0,Y 36.06,Z 468.457,A -85,B 0,C 180,E1 -29947.048,E2 -29947.048} C_VEL
LIN {X 0,Y 34.484,Z 470.771,A -85,B 0,C 180,E1 -29958.231,E2 -29958.231} C_VEL
LIN {X 0,Y 34.122,Z 472.643,A -85,B 0,C 180,E1 -29969.99,E2 -29969.99} C_VEL
LIN {X 0,Y 34.502,Z 474.031,A -85,B 0,C 180,E1 -29981.743,E2 -29981.743} C_VEL
LIN {X 0,Y 38.842,Z 475.614,A -85,B 0,C 180,E1 -30002.865,E2 -30002.865} C_VEL
LIN {X 0,Y 46.982,Z 475.72,A -85,B 0,C 180,E1 -30018.401,E2 -30018.401} C_VEL
LIN {X 0,Y 57.611,Z 474.275,A -85,B 0,C 180,E1 -30028.631,E2 -30028.631} C_VEL
LIN {X 0,Y 69.5,Z 471.318,A -85,B 0,C 180,E1 -30035.507,E2 -30035.507} C_VEL
LIN {X 0,Y 78.86,Z 468.009,A -85,B 0,C 180,E1 -30039.338,E2 -30039.338} C_VEL
LIN {X 0,Y 88.534,Z 463.689,A -85,B 0,C 180,E1 -30042.271,E2 -30042.271} C_VEL
LIN {X 0,Y 100.097,Z 457.219,A -85,B 0,C 180,E1 -30044.873,E2 -30044.873} C_VEL
LIN {X 0,Y 108.45,Z 451.484,A -85,B 0,C 180,E1 -30046.409,E2 -30046.409} C_VEL
LIN {X 0,Y 116.897,Z 444.619,A -85,B 0,C 180,E1 -30047.665,E2 -30047.665} C_VEL
LIN {X 0,Y 123.418,Z 438.428,A -85,B 0,C 180,E1 -30048.462,E2 -30048.462} C_VEL
LIN {X 0,Y 124.043,Z 437.776,A -85,B 0,C 180,E1 -30049.028,E2 -30049.028} C_VEL
LIN {X 0,Y 114.029,Z 447.018,A -85,B 0,C 180,E1 -30050.427,E2 -30050.427} C_VEL
LIN {X 0,Y 103.487,Z 454.869,A -85,B 0,C 180,E1 -30052.181,E2 -30052.181} C_VEL
LIN {X 0,Y 91.744,Z 461.836,A -85,B 0,C 180,E1 -30054.736,E2 -30054.736} C_VEL
LIN {X 0,Y 80.87,Z 466.917,A -85,B 0,C 180,E1 -30057.891,E2 -30057.891} C_VEL
LIN {X 0,Y 78.909,Z 467.672,A -85,B 0,C 180,E1 -30058.569,E2 -30058.569} C_VEL
LIN {X 0,Y 73.632,Z 469.573,A -85,B 0,C 180,E1 -30060.008,E2 -30060.008} C_VEL
LIN {X 0,Y 64.221,Z 472.181,A -85,B 0,C 180,E1 -30061.476,E2 -30061.476} C_VEL
LIN {X 0,Y 54.727,Z 474.04,A -85,B 0,C 180,E1 -30063.532,E2 -30063.532} C_VEL
LIN {X 0,Y 49.448,Z 474.689,A -85,B 0,C 180,E1 -30066.342,E2 -30066.342} C_VEL
LIN {X 0,Y 43.122,Z 475.168,A -85,B 0,C 180,E1 -30072.115,E2 -30072.115} C_VEL
LIN {X 0,Y 35.262,Z 475.069,A -85,B 0,C 180,E1 -30083.449,E2 -30083.449} C_VEL
LIN {X 0,Y 28.644,Z 473.803,A -85,B 0,C 180,E1 -30102.621,E2 -30102.621} C_VEL
LIN {X 0,Y 26.583,Z 472.405,A -85,B 0,C 180,E1 -30118.093,E2 -30118.093} C_VEL
LIN {X 0,Y 27.228,Z 469.438,A -85,B 0,C 180,E1 -30142.473,E2 -30142.473} C_VEL
LIN {X 0,Y 31.715,Z 465.315,A -85,B 0,C 180,E1 -30162.813,E2 -30162.813} C_VEL
LIN {X 0,Y 38.781,Z 459.815,A -85,B 0,C 180,E1 -30177.533,E2 -30177.533} C_VEL
LIN {X 0,Y 46.795,Z 453.28,A -85,B 0,C 180,E1 -30186.932,E2 -30186.932} C_VEL
LIN {X 0,Y 55.887,Z 444.861,A -85,B 0,C 180,E1 -30193.768,E2 -30193.768} C_VEL
LIN {X 0,Y 64.514,Z 435.51,A -85,B 0,C 180,E1 -30198.213,E2 -30198.213} C_VEL
LIN {X 0,Y 72.138,Z 425.523,A -85,B 0,C 180,E1 -30201.212,E2 -30201.212} C_VEL
LIN {X 0,Y 78.872,Z 414.864,A -85,B 0,C 180,E1 -30203.324,E2 -30203.324} C_VEL
LIN {X 0,Y 84.811,Z 403.177,A -85,B 0,C 180,E1 -30204.922,E2 -30204.922} C_VEL
LIN {X 0,Y 89.401,Z 391.29,A -85,B 0,C 180,E1 -30206.089,E2 -30206.089} C_VEL
LIN {X 0,Y 93.175,Z 377.813,A -85,B 0,C 180,E1 -30206.91,E2 -30206.91} C_VEL
LIN {X 0,Y 95.547,Z 364.108,A -85,B 0,C 180,E1 -30207.394,E2 -30207.394} C_VEL
LIN {X 0,Y 96.02,Z 359.807,A -85,B 0,C 180,E1 -30207.614,E2 -30207.614} C_VEL
LIN {X 0,Y 94.559,Z 355.156,A -85,B 0,C 180,E1 -30211.578,E2 -30211.578} C_VEL
LIN {X 0,Y 93.322,Z 351.308,A -85,B 0,C 180,E1 -30216.051,E2 -30216.051} C_VEL
LIN {X 0,Y 92.381,Z 348.545,A -85,B 0,C 180,E1 -30220.924,E2 -30220.924} C_VEL
LIN {X 0,Y 91.969,Z 346.309,A -85,B 0,C 180,E1 -30229.448,E2 -30229.448} C_VEL
LIN {X 0,Y 92.127,Z 346.665,A -85,B 0,C 180,E1 -30232.645,E2 -30232.645} C_VEL
LIN {X 0,Y 92.692,Z 348.703,A -85,B 0,C 180,E1 -30237.379,E2 -30237.379} C_VEL
LIN {X 0,Y 93.53,Z 351.689,A -85,B 0,C 180,E1 -30241.557,E2 -30241.557} C_VEL
LIN {X 0,Y 94.818,Z 355.688,A -85,B 0,C 180,E1 -30245.944,E2 -30245.944} C_VEL
LIN {X 0,Y 96.1,Z 359.905,A -85,B 0,C 180,E1 -30249.361,E2 -30249.361} C_VEL
LIN {X 0,Y 93.764,Z 375.957,A -85,B 0,C 180,E1 -30249.984,E2 -30249.984} C_VEL
LIN {X 0,Y 90.66,Z 388.075,A -85,B 0,C 180,E1 -30250.525,E2 -30250.525} C_VEL
LIN {X 0,Y 86.781,Z 399.088,A -85,B 0,C 180,E1 -30251.369,E2 -30251.369} C_VEL
LIN {X 0,Y 81.068,Z 411.393,A -85,B 0,C 180,E1 -30252.746,E2 -30252.746} C_VEL
LIN {X 0,Y 75.269,Z 421.365,A -85,B 0,C 180,E1 -30254.348,E2 -30254.348} C_VEL
LIN {X 0,Y 67.949,Z 431.815,A -85,B 0,C 180,E1 -30256.901,E2 -30256.901} C_VEL
LIN {X 0,Y 59.332,Z 441.932,A -85,B 0,C 180,E1 -30260.839,E2 -30260.839} C_VEL
LIN {X 0,Y 50.887,Z 450.275,A -85,B 0,C 180,E1 -30266.127,E2 -30266.127} C_VEL
LIN {X 0,Y 42.44,Z 457.571,A -85,B 0,C 180,E1 -30274.094,E2 -30274.094} C_VEL
LIN {X 0,Y 35.021,Z 463.359,A -85,B 0,C 180,E1 -30285.369,E2 -30285.369} C_VEL
LIN {X 0,Y 29.64,Z 467.907,A -85,B 0,C 180,E1 -30301.679,E2 -30301.679} C_VEL
LIN {X 0,Y 27.565,Z 470.283,A -85,B 0,C 180,E1 -30315.216,E2 -30315.216} C_VEL
LIN {X 0,Y 27.031,Z 472.217,A -85,B 0,C 180,E1 -30329.988,E2 -30329.988} C_VEL
LIN {X 0,Y 27.603,Z 473.705,A -85,B 0,C 180,E1 -30344.738,E2 -30344.738} C_VEL
LIN {X 0,Y 29.687,Z 474.763,A -85,B 0,C 180,E1 -30358.247,E2 -30358.247} C_VEL
LIN {X 0,Y 37.466,Z 475.722,A -85,B 0,C 180,E1 -30378.606,E2 -30378.606} C_VEL
LIN {X 0,Y 48.264,Z 475.223,A -85,B 0,C 180,E1 -30390.876,E2 -30390.876} C_VEL
LIN {X 0,Y 60.47,Z 473.171,A -85,B 0,C 180,E1 -30398.386,E2 -30398.386} C_VEL
LIN {X 0,Y 73.357,Z 469.579,A -85,B 0,C 180,E1 -30403.329,E2 -30403.329} C_VEL
LIN {X 0,Y 83.288,Z 465.742,A -85,B 0,C 180,E1 -30406.006,E2 -30406.006} C_VEL
LIN {X 0,Y 93.39,Z 460.834,A -85,B 0,C 180,E1 -30408.023,E2 -30408.023} C_VEL
LIN {X 0,Y 96.135,Z 459.285,A -85,B 0,C 180,E1 -30409.311,E2 -30409.311} C_VEL
LIN {X 0,Y 85.279,Z 464.781,A -85,B 0,C 180,E1 -30411.442,E2 -30411.442} C_VEL
LIN {X 0,Y 73.688,Z 469.303,A -85,B 0,C 180,E1 -30414.509,E2 -30414.509} C_VEL
LIN {X 0,Y 59.682,Z 473.066,A -85,B 0,C 180,E1 -30419.977,E2 -30419.977} C_VEL
LIN {X 0,Y 49.448,Z 474.689,A -85,B 0,C 180,E1 -30426.342,E2 -30426.342} C_VEL
LIN {X 0,Y 44.278,Z 475.116,A -85,B 0,C 180,E1 -30429.831,E2 -30429.831} C_VEL
LIN {X 0,Y 35.099,Z 475.209,A -85,B 0,C 180,E1 -30435.329,E2 -30435.329} C_VEL
LIN {X 0,Y 27.994,Z 474.744,A -85,B 0,C 180,E1 -30441.908,E2 -30441.908} C_VEL
LIN {X 0,Y 23.577,Z 474.037,A -85,B 0,C 180,E1 -30450.638,E2 -30450.638} C_VEL
LIN {X 0,Y 22.466,Z 473.712,A -85,B 0,C 180,E1 -30454.655,E2 -30454.655} C_VEL
LIN {X 0,Y 19.196,Z 471.099,A -85,B 0,C 180,E1 -30488.542,E2 -30488.542} C_VEL
LIN {X 0,Y 22.589,Z 467.409,A -85,B 0,C 180,E1 -30519.824,E2 -30519.824} C_VEL
LIN {X 0,Y 29.368,Z 462.819,A -85,B 0,C 180,E1 -30538.608,E2 -30538.608} C_VEL
LIN {X 0,Y 38.235,Z 456.648,A -85,B 0,C 180,E1 -30550.515,E2 -30550.515} C_VEL
LIN {X 0,Y 47.552,Z 449.227,A -85,B 0,C 180,E1 -30557.655,E2 -30557.655} C_VEL
LIN {X 0,Y 56.807,Z 440.534,A -85,B 0,C 180,E1 -30562.248,E2 -30562.248} C_VEL
LIN {X 0,Y 65.205,Z 431.022,A -85,B 0,C 180,E1 -30565.278,E2 -30565.278} C_VEL
LIN {X 0,Y 72.96,Z 420.262,A -85,B 0,C 180,E1 -30567.451,E2 -30567.451} C_VEL
LIN {X 0,Y 79.966,Z 408.235,A -85,B 0,C 180,E1 -30568.978,E2 -30568.978} C_VEL
LIN {X 0,Y 85.209,Z 396.463,A -85,B 0,C 180,E1 -30570.077,E2 -30570.077} C_VEL
LIN {X 0,Y 89.639,Z 383.084,A -85,B 0,C 180,E1 -30570.871,E2 -30570.871} C_VEL
LIN {X 0,Y 92.456,Z 370.315,A -85,B 0,C 180,E1 -30571.359,E2 -30571.359} C_VEL
LIN {X 0,Y 93.43,Z 363.66,A -85,B 0,C 180,E1 -30571.488,E2 -30571.488} C_VEL
LIN {X 0,Y 93.214,Z 362.526,A -85,B 0,C 180,E1 -30572.315,E2 -30572.315} C_VEL
LIN {X 0,Y 92.106,Z 358.318,A -85,B 0,C 180,E1 -30576.911,E2 -30576.911} C_VEL
LIN {X 0,Y 91.257,Z 355.377,A -85,B 0,C 180,E1 -30582.075,E2 -30582.075} C_VEL
LIN {X 0,Y 91.031,Z 353.365,A -85,B 0,C 180,E1 -30589.338,E2 -30589.338} C_VEL
LIN {X 0,Y 91.127,Z 353.608,A -85,B 0,C 180,E1 -30591.854,E2 -30591.854} C_VEL
LIN {X 0,Y 91.497,Z 355.362,A -85,B 0,C 180,E1 -30596.029,E2 -30596.029} C_VEL
LIN {X 0,Y 92.399,Z 359.093,A -85,B 0,C 180,E1 -30601.186,E2 -30601.186} C_VEL
LIN {X 0,Y 93.496,Z 363.361,A -85,B 0,C 180,E1 -30605.394,E2 -30605.394} C_VEL
LIN {X 0,Y 91.404,Z 376.519,A -85,B 0,C 180,E1 -30605.842,E2 -30605.842} C_VEL
LIN {X 0,Y 88.23,Z 388.425,A -85,B 0,C 180,E1 -30606.252,E2 -30606.252} C_VEL
LIN {X 0,Y 84.078,Z 399.731,A -85,B 0,C 180,E1 -30606.934,E2 -30606.934} C_VEL
LIN {X 0,Y 78.093,Z 412.162,A -85,B 0,C 180,E1 -30608.105,E2 -30608.105} C_VEL
LIN {X 0,Y 72.12,Z 421.957,A -85,B 0,C 180,E1 -30609.342,E2 -30609.342} C_VEL
LIN {X 0,Y 64.546,Z 432.283,A -85,B 0,C 180,E1 -30611.467,E2 -30611.467} C_VEL
LIN {X 0,Y 56.519,Z 441.305,A -85,B 0,C 180,E1 -30614.425,E2 -30614.425} C_VEL
LIN {X 0,Y 48.178,Z 449.182,A -85,B 0,C 180,E1 -30618.505,E2 -30618.505} C_VEL
LIN {X 0,Y 38.881,Z 456.646,A -85,B 0,C 180,E1 -30625.322,E2 -30625.322} C_VEL
LIN {X 0,Y 30.361,Z 462.609,A -85,B 0,C 180,E1 -30635.868,E2 -30635.868} C_VEL
LIN {X 0,Y 23.626,Z 467.309,A -85,B 0,C 180,E1 -30653.475,E2 -30653.475} C_VEL
LIN {X 0,Y 20.062,Z 470.852,A -85,B 0,C 180,E1 -30679.895,E2 -30679.895} C_VEL
LIN {X 0,Y 19.951,Z 471.792,A -85,B 0,C 180,E1 -30689.983,E2 -30689.983} C_VEL
LIN {X 0,Y 20.81,Z 473.34,A -85,B 0,C 180,E1 -30709.721,E2 -30709.721} C_VEL
LIN {X 0,Y 23.669,Z 474.493,A -85,B 0,C 180,E1 -30726.414,E2 -30726.414} C_VEL
LIN {X 0,Y 33.184,Z 475.592,A -85,B 0,C 180,E1 -30747.885,E2 -30747.885} C_VEL
LIN {X 0,Y 45.233,Z 475.221,A -85,B 0,C 180,E1 -30758.764,E2 -30758.764} C_VEL
LIN {X 0,Y 51.648,Z 474.49,A -85,B 0,C 180,E1 -30762.251,E2 -30762.251} C_VEL
LIN {X 0,Y 64.909,Z 471.822,A -85,B 0,C 180,E1 -30767.002,E2 -30767.002} C_VEL
LIN {X 0,Y 71.644,Z 469.898,A -85,B 0,C 180,E1 -30768.776,E2 -30768.776} C_VEL
LIN {X 0,Y 71.543,Z 469.921,A -85,B 0,C 180,E1 -30769.189,E2 -30769.189} C_VEL
LIN {X 0,Y 58.345,Z 473.228,A -85,B 0,C 180,E1 -30773.058,E2 -30773.058} C_VEL
